LIN {X 0,Y 117.836,Z 740.059,A -85,B 0,C 180,E1 -26007.711,E2 -26007.711} C_VEL
LIN {X 0,Y 116.327,Z 745.047,A -85,B 0,C 180,E1 -26011.731,E2 -26011.731} C_VEL
LIN {X 0,Y 115.88,Z 750.752,A -85,B 0,C 180,E1 -26016.967,E2 -26016.967} C_VEL
LIN {X 0,Y 115.857,Z 756.729,A -85,B 0,C 180,E1 -26024.043,E2 -26024.043} C_VEL
LIN {X 0,Y 117.699,Z 761.437,A -85,B 0,C 180,E1 -26030.994,E2 -26030.994} C_VEL
LIN {X 0,Y 121.56,Z 765.132,A -85,B 0,C 180,E1 -26037.55,E2 -26037.55} C_VEL
LIN {X 0,Y 129.441,Z 768.589,A -85,B 0,C 180,E1 -26045.469,E2 -26045.469} C_VEL
LIN {X 0,Y 138.496,Z 770.335,A -85,B 0,C 180,E1 -26051.277,E2 -26051.277} C_VEL
LIN {X 0,Y 147.642,Z 770.918,A -85,B 0,C 180,E1 -26055.564,E2 -26055.564} C_VEL
LIN {X 0,Y 151.092,Z 770.908,A -85,B 0,C 180,E1 -26056.893,E2 -26056.893} C_VEL
LIN {X 0,Y 151.584,Z 770.825,A -85,B 0,C 180,E1 -26057.685,E2 -26057.685} C_VEL
LIN {X 0,Y 144.117,Z 770,A -85,B 0,C 180,E1 -26060.657,E2 -26060.657} C_VEL
LIN {X 0,Y 136.812,Z 768.361,A -85,B 0,C 180,E1 -26064.334,E2 -26064.334} C_VEL
LIN {X 0,Y 132.911,Z 767.253,A -85,B 0,C 180,E1 -26066.154,E2 -26066.154} C_VEL
LIN {X 0,Y 125.626,Z 764.718,A -85,B 0,C 180,E1 -26068.907,E2 -26068.907} C_VEL
LIN {X 0,Y 118.967,Z 761.486,A -85,B 0,C 180,E1 -26071.986,E2 -26071.986} C_VEL
LIN {X 0,Y 116.161,Z 759.416,A -85,B 0,C 180,E1 -26074.303,E2 -26074.303} C_VEL
LIN {X 0,Y 111.413,Z 753.187,A -85,B 0,C 180,E1 -26081.615,E2 -26081.615} C_VEL
LIN {X 0,Y 108.838,Z 744.994,A -85,B 0,C 180,E1 -26089.771,E2 -26089.771} C_VEL
LIN {X 0,Y 108.339,Z 738.209,A -85,B 0,C 180,E1 -26095.349,E2 -26095.349} C_VEL
LIN {X 0,Y 108.225,Z 729.961,A -85,B 0,C 180,E1 -26100.93,E2 -26100.93} C_VEL
LIN {X 0,Y 108.303,Z 721.553,A -85,B 0,C 180,E1 -26105.586,E2 -26105.586} C_VEL
LIN {X 0,Y 108.9,Z 710.32,A -85,B 0,C 180,E1 -26110.693,E2 -26110.693} C_VEL
LIN {X 0,Y 109.945,Z 696.049,A -85,B 0,C 180,E1 -26115.859,E2 -26115.859} C_VEL
LIN {X 0,Y 111.19,Z 683.821,A -85,B 0,C 180,E1 -26119.38,E2 -26119.38} C_VEL
LIN {X 0,Y 112.386,Z 671.062,A -85,B 0,C 180,E1 -26122.279,E2 -26122.279} C_VEL
LIN {X 0,Y 113.626,Z 656.475,A -85,B 0,C 180,E1 -26124.799,E2 -26124.799} C_VEL
LIN {X 0,Y 117.508,Z 604.417,A -85,B 0,C 180,E1 -26131.43,E2 -26131.43} C_VEL
LIN {X 0,Y 118.923,Z 587.439,A -85,B 0,C 180,E1 -26133.466,E2 -26133.466} C_VEL
LIN {X 0,Y 117.065,Z 560.293,A -85,B 0,C 180,E1 -26136.871,E2 -26136.871} C_VEL
LIN {X 0,Y 110.897,Z 536.307,A -85,B 0,C 180,E1 -26140.492,E2 -26140.492} C_VEL
LIN {X 0,Y 108.832,Z 527.055,A -85,B 0,C 180,E1 -26147.308,E2 -26147.308} C_VEL
LIN {X 0,Y 107.788,Z 522.184,A -85,B 0,C 180,E1 -26151.2,E2 -26151.2} C_VEL
LIN {X 0,Y 107.799,Z 522.181,A -85,B 0,C 180,E1 -26158.562,E2 -26158.562} C_VEL
LIN {X 0,Y 107.912,Z 522.166,A -85,B 0,C 180,E1 -26166.998,E2 -26166.998} C_VEL
LIN {X 0,Y 108.041,Z 522.149,A -85,B 0,C 180,E1 -26174.918,E2 -26174.918} C_VEL
LIN {X 0,Y 108.308,Z 522.117,A -85,B 0,C 180,E1 -26178.774,E2 -26178.774} C_VEL
LIN {X 0,Y 108.466,Z 522.098,A -85,B 0,C 180,E1 -26186.285,E2 -26186.285} C_VEL
LIN {X 0,Y 108.949,Z 522.032,A -85,B 0,C 180,E1 -26190,E2 -26190} C_VEL
LIN {X 0,Y 108.342,Z 522.108,A -85,B 0,C 180,E1 -26197.454,E2 -26197.454} C_VEL
LIN {X 0,Y 108.204,Z 522.132,A -85,B 0,C 180,E1 -26203.026,E2 -26203.026} C_VEL
LIN {X 0,Y 107.911,Z 522.165,A -85,B 0,C 180,E1 -26209.004,E2 -26209.004} C_VEL
LIN {X 0,Y 107.858,Z 522.169,A -85,B 0,C 180,E1 -26214.184,E2 -26214.184} C_VEL
LIN {X 0,Y 107.795,Z 522.179,A -85,B 0,C 180,E1 -26222.052,E2 -26222.052} C_VEL
LIN {X 0,Y 107.715,Z 522.192,A -85,B 0,C 180,E1 -26228.468,E2 -26228.468} C_VEL
LIN {X 0,Y 107.852,Z 522.23,A -85,B 0,C 180,E1 -26233.59,E2 -26233.59} C_VEL
LIN {X 0,Y 111.116,Z 536.487,A -85,B 0,C 180,E1 -26240.246,E2 -26240.246} C_VEL
LIN {X 0,Y 114.313,Z 550.66,A -85,B 0,C 180,E1 -26246.405,E2 -26246.405} C_VEL
LIN {X 0,Y 114.295,Z 554.161,A -85,B 0,C 180,E1 -26247.728,E2 -26247.728} C_VEL
LIN {X 0,Y 115.295,Z 578.296,A -85,B 0,C 180,E1 -26250.622,E2 -26250.622} C_VEL
LIN {X 0,Y 116.148,Z 589.056,A -85,B 0,C 180,E1 -26251.911,E2 -26251.911} C_VEL
LIN {X 0,Y 112.728,Z 655.949,A -85,B 0,C 180,E1 -26260.525,E2 -26260.525} C_VEL
LIN {X 0,Y 111.929,Z 671.773,A -85,B 0,C 180,E1 -26262.883,E2 -26262.883} C_VEL
LIN {X 0,Y 111.129,Z 684.001,A -85,B 0,C 180,E1 -26265.347,E2 -26265.347} C_VEL
LIN {X 0,Y 110.258,Z 697.634,A -85,B 0,C 180,E1 -26268.976,E2 -26268.976} C_VEL
LIN {X 0,Y 109.668,Z 708.586,A -85,B 0,C 180,E1 -26272.636,E2 -26272.636} C_VEL
LIN {X 0,Y 109.307,Z 719.724,A -85,B 0,C 180,E1 -26277.236,E2 -26277.236} C_VEL
LIN {X 0,Y 109.26,Z 728.724,A -85,B 0,C 180,E1 -26281.843,E2 -26281.843} C_VEL
LIN {X 0,Y 109.364,Z 736.128,A -85,B 0,C 180,E1 -26286.457,E2 -26286.457} C_VEL
LIN {X 0,Y 109.683,Z 743.345,A -85,B 0,C 180,E1 -26292.02,E2 -26292.02} C_VEL
LIN {X 0,Y 111.458,Z 750.421,A -85,B 0,C 180,E1 -26298.378,E2 -26298.378} C_VEL
LIN {X 0,Y 115.207,Z 756.964,A -85,B 0,C 180,E1 -26305.279,E2 -26305.279} C_VEL
LIN {X 0,Y 120.801,Z 762.203,A -85,B 0,C 180,E1 -26311.574,E2 -26311.574} C_VEL
LIN {X 0,Y 128.236,Z 766.306,A -85,B 0,C 180,E1 -26317.075,E2 -26317.075} C_VEL
LIN {X 0,Y 137.135,Z 769.302,A -85,B 0,C 180,E1 -26321.777,E2 -26321.777} C_VEL
LIN {X 0,Y 140.576,Z 770.083,A -85,B 0,C 180,E1 -26323.232,E2 -26323.232} C_VEL
LIN {X 0,Y 140.221,Z 770.131,A -85,B 0,C 180,E1 -26324.287,E2 -26324.287} C_VEL
LIN {X 0,Y 129.693,Z 768.061,A -85,B 0,C 180,E1 -26329.438,E2 -26329.438} C_VEL
LIN {X 0,Y 122.094,Z 765.265,A -85,B 0,C 180,E1 -26334.857,E2 -26334.857} C_VEL
LIN {X 0,Y 116.195,Z 761.467,A -85,B 0,C 180,E1 -26341.061,E2 -26341.061} C_VEL
LIN {X 0,Y 112.25,Z 756.576,A -85,B 0,C 180,E1 -26347.935,E2 -26347.935} C_VEL
LIN {X 0,Y 110.479,Z 750.464,A -85,B 0,C 180,E1 -26355.259,E2 -26355.259} C_VEL
LIN {X 0,Y 110.594,Z 743.772,A -85,B 0,C 180,E1 -26361.78,E2 -26361.78} C_VEL
LIN {X 0,Y 111.699,Z 736.584,A -85,B 0,C 180,E1 -26367.45,E2 -26367.45} C_VEL
LIN {X 0,Y 109.948,Z 741.833,A -85,B 0,C 180,E1 -26371.832,E2 -26371.832} C_VEL
LIN {X 0,Y 109.438,Z 747.875,A -85,B 0,C 180,E1 -26377.38,E2 -26377.38} C_VEL
LIN {X 0,Y 109.482,Z 754.136,A -85,B 0,C 180,E1 -26384.879,E2 -26384.879} C_VEL
LIN {X 0,Y 111.446,Z 759.184,A -85,B 0,C 180,E1 -26392.233,E2 -26392.233} C_VEL
LIN {X 0,Y 115.538,Z 763.209,A -85,B 0,C 180,E1 -26399.119,E2 -26399.119} C_VEL
LIN {X 0,Y 121.444,Z 766.263,A -85,B 0,C 180,E1 -26405.36,E2 -26405.36} C_VEL
LIN {X 0,Y 129.062,Z 768.493,A -85,B 0,C 180,E1 -26410.803,E2 -26410.803} C_VEL
LIN {X 0,Y 139.931,Z 770.054,A -85,B 0,C 180,E1 -26416.427,E2 -26416.427} C_VEL
LIN {X 0,Y 141.036,Z 770.146,A -85,B 0,C 180,E1 -26416.878,E2 -26416.878} C_VEL
LIN {X 0,Y 140.5,Z 769.925,A -85,B 0,C 180,E1 -26418.058,E2 -26418.058} C_VEL
LIN {X 0,Y 129.613,Z 767.124,A -85,B 0,C 180,E1 -26423.384,E2 -26423.384} C_VEL
LIN {X 0,Y 120.074,Z 762.583,A -85,B 0,C 180,E1 -26430.164,E2 -26430.164} C_VEL
LIN {X 0,Y 116.161,Z 759.416,A -85,B 0,C 180,E1 -26434.303,E2 -26434.303} C_VEL
LIN {X 0,Y 113.641,Z 757.196,A -85,B 0,C 180,E1 -26436.712,E2 -26436.712} C_VEL
LIN {X 0,Y 106.531,Z 750.669,A -85,B 0,C 180,E1 -26441.919,E2 -26441.919} C_VEL
LIN {X 0,Y 103.471,Z 746.464,A -85,B 0,C 180,E1 -26445.213,E2 -26445.213} C_VEL
LIN {X 0,Y 102.733,Z 744.402,A -85,B 0,C 180,E1 -26447.052,E2 -26447.052} C_VEL
LIN {X 0,Y 101.854,Z 736.413,A -85,B 0,C 180,E1 -26454.059,E2 -26454.059} C_VEL
LIN {X 0,Y 101.623,Z 729.435,A -85,B 0,C 180,E1 -26459.009,E2 -26459.009} C_VEL
LIN {X 0,Y 101.655,Z 721.117,A -85,B 0,C 180,E1 -26463.964,E2 -26463.964} C_VEL
LIN {X 0,Y 102.025,Z 710.024,A -85,B 0,C 180,E1 -26469.416,E2 -26469.416} C_VEL
LIN {X 0,Y 102.767,Z 697.76,A -85,B 0,C 180,E1 -26474.209,E2 -26474.209} C_VEL
LIN {X 0,Y 103.928,Z 686.164,A -85,B 0,C 180,E1 -26477.938,E2 -26477.938} C_VEL
LIN {X 0,Y 105.202,Z 672.771,A -85,B 0,C 180,E1 -26481.351,E2 -26481.351} C_VEL
LIN {X 0,Y 106.464,Z 657.142,A -85,B 0,C 180,E1 -26484.367,E2 -26484.367} C_VEL
LIN {X 0,Y 109.13,Z 620.339,A -85,B 0,C 180,E1 -26489.542,E2 -26489.542} C_VEL
LIN {X 0,Y 111.81,Z 587.596,A -85,B 0,C 180,E1 -26493.772,E2 -26493.772} C_VEL
LIN {X 0,Y 110.129,Z 561.697,A -85,B 0,C 180,E1 -26497.239,E2 -26497.239} C_VEL
LIN {X 0,Y 103.597,Z 536.147,A -85,B 0,C 180,E1 -26501.368,E2 -26501.368} C_VEL
LIN {X 0,Y 101.86,Z 528.349,A -85,B 0,C 180,E1 -26507.502,E2 -26507.502} C_VEL
LIN {X 0,Y 100.703,Z 523.066,A -85,B 0,C 180,E1 -26512.046,E2 -26512.046} C_VEL
LIN {X 0,Y 100.693,Z 523.062,A -85,B 0,C 180,E1 -26516.882,E2 -26516.882} C_VEL
LIN {X 0,Y 100.787,Z 523.049,A -85,B 0,C 180,E1 -26525.267,E2 -26525.267} C_VEL
LIN {X 0,Y 100.82,Z 523.051,A -85,B 0,C 180,E1 -26529.601,E2 -26529.601} C_VEL
LIN {X 0,Y 101.2,Z 523.003,A -85,B 0,C 180,E1 -26537.975,E2 -26537.975} C_VEL
LIN {X 0,Y 101.281,Z 522.988,A -85,B 0,C 180,E1 -26542.022,E2 -26542.022} C_VEL
LIN {X 0,Y 101.873,Z 522.913,A -85,B 0,C 180,E1 -26550,E2 -26550} C_VEL
LIN {X 0,Y 101.281,Z 522.986,A -85,B 0,C 180,E1 -26557.977,E2 -26557.977} C_VEL
LIN {X 0,Y 101.13,Z 523.013,A -85,B 0,C 180,E1 -26563.363,E2 -26563.363} C_VEL
LIN {X 0,Y 100.82,Z 523.051,A -85,B 0,C 180,E1 -26570.398,E2 -26570.398} C_VEL
LIN {X 0,Y 100.775,Z 523.05,A -85,B 0,C 180,E1 -26574.958,E2 -26574.958} C_VEL
LIN {X 0,Y 100.701,Z 523.06,A -85,B 0,C 180,E1 -26583.124,E2 -26583.124} C_VEL
LIN {X 0,Y 100.739,Z 523.053,A -85,B 0,C 180,E1 -26591.798,E2 -26591.798} C_VEL
LIN {X 0,Y 100.813,Z 523.12,A -85,B 0,C 180,E1 -26592.967,E2 -26592.967} C_VEL
LIN {X 0,Y 104.128,Z 537.755,A -85,B 0,C 180,E1 -26600.152,E2 -26600.152} C_VEL
LIN {X 0,Y 107.067,Z 550.686,A -85,B 0,C 180,E1 -26606.088,E2 -26606.088} C_VEL
LIN {X 0,Y 107.21,Z 553.958,A -85,B 0,C 180,E1 -26607.472,E2 -26607.472} C_VEL
LIN {X 0,Y 108.263,Z 579.215,A -85,B 0,C 180,E1 -26610.75,E2 -26610.75} C_VEL
LIN {X 0,Y 108.966,Z 589.885,A -85,B 0,C 180,E1 -26612.121,E2 -26612.121} C_VEL
LIN {X 0,Y 105.725,Z 658.101,A -85,B 0,C 180,E1 -26621.594,E2 -26621.594} C_VEL
LIN {X 0,Y 104.911,Z 673.601,A -85,B 0,C 180,E1 -26624.208,E2 -26624.208} C_VEL
LIN {X 0,Y 104.067,Z 687.071,A -85,B 0,C 180,E1 -26627.321,E2 -26627.321} C_VEL
LIN {X 0,Y 103.38,Z 700.092,A -85,B 0,C 180,E1 -26631.202,E2 -26631.202} C_VEL
LIN {X 0,Y 102.914,Z 710.414,A -85,B 0,C 180,E1 -26635.103,E2 -26635.103} C_VEL
LIN {X 0,Y 102.837,Z 721.004,A -85,B 0,C 180,E1 -26640,E2 -26640} C_VEL
LIN {X 0,Y 102.956,Z 729.651,A -85,B 0,C 180,E1 -26644.895,E2 -26644.895} C_VEL
LIN {X 0,Y 103.139,Z 736.605,A -85,B 0,C 180,E1 -26649.808,E2 -26649.808} C_VEL
LIN {X 0,Y 104.524,Z 745.743,A -85,B 0,C 180,E1 -26657.612,E2 -26657.612} C_VEL
LIN {X 0,Y 107.965,Z 753.091,A -85,B 0,C 180,E1 -26665.032,E2 -26665.032} C_VEL
LIN {X 0,Y 113.43,Z 759.062,A -85,B 0,C 180,E1 -26671.779,E2 -26671.779} C_VEL
LIN {X 0,Y 120.684,Z 763.854,A -85,B 0,C 180,E1 -26677.696,E2 -26677.696} C_VEL
LIN {X 0,Y 130.665,Z 767.952,A -85,B 0,C 180,E1 -26683.202,E2 -26683.202} C_VEL
LIN {X 0,Y 130.428,Z 768.003,A -85,B 0,C 180,E1 -26684.327,E2 -26684.327} C_VEL
LIN {X 0,Y 124.527,Z 766.414,A -85,B 0,C 180,E1 -26687.371,E2 -26687.371} C_VEL
LIN {X 0,Y 116.607,Z 763.235,A -85,B 0,C 180,E1 -26692.936,E2 -26692.936} C_VEL
LIN {X 0,Y 110.417,Z 759.069,A -85,B 0,C 180,E1 -26699.39,E2 -26699.39} C_VEL
LIN {X 0,Y 106.233,Z 753.781,A -85,B 0,C 180,E1 -26706.613,E2 -26706.613} C_VEL
LIN {X 0,Y 104.358,Z 747.267,A -85,B 0,C 180,E1 -26714.373,E2 -26714.373} C_VEL
LIN {X 0,Y 104.382,Z 741.354,A -85,B 0,C 180,E1 -26720.31,E2 -26720.31} C_VEL
LIN {X 0,Y 105.663,Z 732.897,A -85,B 0,C 180,E1 -26727.248,E2 -26727.248} C_VEL
LIN {X 0,Y 103.663,Z 738.443,A -85,B 0,C 180,E1 -26731.943,E2 -26731.943} C_VEL
LIN {X 0,Y 103.087,Z 744.796,A -85,B 0,C 180,E1 -26737.837,E2 -26737.837} C_VEL
LIN {X 0,Y 103.171,Z 751.383,A -85,B 0,C 180,E1 -26745.812,E2 -26745.812} C_VEL
LIN {X 0,Y 105.317,Z 756.697,A -85,B 0,C 180,E1 -26753.603,E2 -26753.603} C_VEL
LIN {X 0,Y 109.681,Z 761.067,A -85,B 0,C 180,E1 -26760.839,E2 -26760.839} C_VEL
LIN {X 0,Y 115.909,Z 764.481,A -85,B 0,C 180,E1 -26767.326,E2 -26767.326} C_VEL
LIN {X 0,Y 123.89,Z 767.035,A -85,B 0,C 180,E1 -26772.902,E2 -26772.902} C_VEL
LIN {X 0,Y 131.226,Z 768.538,A -85,B 0,C 180,E1 -26776.85,E2 -26776.85} C_VEL
LIN {X 0,Y 130.525,Z 768.205,A -85,B 0,C 180,E1 -26778.142,E2 -26778.142} C_VEL
LIN {X 0,Y 119.793,Z 764.229,A -85,B 0,C 180,E1 -26784.078,E2 -26784.078} C_VEL
LIN {X 0,Y 112.489,Z 759.76,A -85,B 0,C 180,E1 -26790.012,E2 -26790.012} C_VEL
LIN {X 0,Y 107.088,Z 754.177,A -85,B 0,C 180,E1 -26796.811,E2 -26796.811} C_VEL
LIN {X 0,Y 103.505,Z 747.281,A -85,B 0,C 180,E1 -26804.24,E2 -26804.24} C_VEL
LIN {X 0,Y 102.733,Z 744.402,A -85,B 0,C 180,E1 -26807.052,E2 -26807.052} C_VEL
LIN {X 0,Y 101.66,Z 741.184,A -85,B 0,C 180,E1 -26809.735,E2 -26809.735} C_VEL
LIN {X 0,Y 99.905,Z 737.51,A -85,B 0,C 180,E1 -26812.19,E2 -26812.19} C_VEL
LIN {X 0,Y 96.165,Z 729.337,A -85,B 0,C 180,E1 -26816.906,E2 -26816.906} C_VEL
LIN {X 0,Y 95.15,Z 725.073,A -85,B 0,C 180,E1 -26819.392,E2 -26819.392} C_VEL
LIN {X 0,Y 95.071,Z 723.636,A -85,B 0,C 180,E1 -26820.254,E2 -26820.254} C_VEL
LIN {X 0,Y 95.168,Z 713.731,A -85,B 0,C 180,E1 -26825.828,E2 -26825.828} C_VEL
LIN {X 0,Y 95.538,Z 703.495,A -85,B 0,C 180,E1 -26830.597,E2 -26830.597} C_VEL
LIN {X 0,Y 96.562,Z 689.721,A -85,B 0,C 180,E1 -26835.839,E2 -26835.839} C_VEL
LIN {X 0,Y 97.905,Z 675.435,A -85,B 0,C 180,E1 -26840.001,E2 -26840.001} C_VEL
LIN {X 0,Y 99.236,Z 659.449,A -85,B 0,C 180,E1 -26843.474,E2 -26843.474} C_VEL
LIN {X 0,Y 101.423,Z 628.397,A -85,B 0,C 180,E1 -26848.309,E2 -26848.309} C_VEL
LIN {X 0,Y 104.746,Z 588.113,A -85,B 0,C 180,E1 -26854.047,E2 -26854.047} C_VEL
LIN {X 0,Y 103.146,Z 562.959,A -85,B 0,C 180,E1 -26857.63,E2 -26857.63} C_VEL
LIN {X 0,Y 96.32,Z 536.044,A -85,B 0,C 180,E1 -26862.261,E2 -26862.261} C_VEL
LIN {X 0,Y 94.467,Z 527.663,A -85,B 0,C 180,E1 -26869.385,E2 -26869.385} C_VEL
LIN {X 0,Y 93.655,Z 523.943,A -85,B 0,C 180,E1 -26872.769,E2 -26872.769} C_VEL
LIN {X 0,Y 93.585,Z 523.952,A -85,B 0,C 180,E1 -26878.285,E2 -26878.285} C_VEL
LIN {X 0,Y 93.67,Z 523.934,A -85,B 0,C 180,E1 -26884.205,E2 -26884.205} C_VEL
LIN {X 0,Y 93.696,Z 523.939,A -85,B 0,C 180,E1 -26887.973,E2 -26887.973} C_VEL
LIN {X 0,Y 94.099,Z 523.889,A -85,B 0,C 180,E1 -26897.052,E2 -26897.052} C_VEL
LIN {X 0,Y 94.213,Z 523.867,A -85,B 0,C 180,E1 -26901.419,E2 -26901.419} C_VEL
LIN {X 0,Y 94.8,Z 523.794,A -85,B 0,C 180,E1 -26910,E2 -26910} C_VEL
LIN {X 0,Y 94.213,Z 523.866,A -85,B 0,C 180,E1 -26918.58,E2 -26918.58} C_VEL
LIN {X 0,Y 94.048,Z 523.894,A -85,B 0,C 180,E1 -26923.721,E2 -26923.721} C_VEL
LIN {X 0,Y 93.696,Z 523.938,A -85,B 0,C 180,E1 -26932.027,E2 -26932.027} C_VEL
LIN {X 0,Y 93.624,Z 523.943,A -85,B 0,C 180,E1 -26936.769,E2 -26936.769} C_VEL
LIN {X 0,Y 93.6,Z 523.944,A -85,B 0,C 180,E1 -26944.316,E2 -26944.316} C_VEL
LIN {X 0,Y 93.719,Z 523.931,A -85,B 0,C 180,E1 -26952.264,E2 -26952.264} C_VEL
LIN {X 0,Y 96.683,Z 537.098,A -85,B 0,C 180,E1 -26959.139,E2 -26959.139} C_VEL
LIN {X 0,Y 99.512,Z 549.365,A -85,B 0,C 180,E1 -26965.153,E2 -26965.153} C_VEL
LIN {X 0,Y 100.183,Z 553.098,A -85,B 0,C 180,E1 -26966.887,E2 -26966.887} C_VEL
LIN {X 0,Y 100.132,Z 554.433,A -85,B 0,C 180,E1 -26967.378,E2 -26967.378} C_VEL
LIN {X 0,Y 101.192,Z 579.73,A -85,B 0,C 180,E1 -26970.863,E2 -26970.863} C_VEL
LIN {X 0,Y 101.869,Z 589.828,A -85,B 0,C 180,E1 -26972.247,E2 -26972.247} C_VEL
LIN {X 0,Y 98.822,Z 657.872,A -85,B 0,C 180,E1 -26982.541,E2 -26982.541} C_VEL
LIN {X 0,Y 98.096,Z 672.774,A -85,B 0,C 180,E1 -26985.213,E2 -26985.213} C_VEL
LIN {X 0,Y 97.309,Z 686.365,A -85,B 0,C 180,E1 -26988.544,E2 -26988.544} C_VEL
LIN {X 0,Y 96.763,Z 699.268,A -85,B 0,C 180,E1 -26992.698,E2 -26992.698} C_VEL
LIN {X 0,Y 96.452,Z 710.8,A -85,B 0,C 180,E1 -26997.39,E2 -26997.39} C_VEL
LIN {X 0,Y 96.505,Z 720.267,A -85,B 0,C 180,E1 -27002.087,E2 -27002.087} C_VEL
LIN {X 0,Y 96.78,Z 728.722,A -85,B 0,C 180,E1 -27007.301,E2 -27007.301} C_VEL
LIN {X 0,Y 97.095,Z 735.657,A -85,B 0,C 180,E1 -27012.542,E2 -27012.542} C_VEL
LIN {X 0,Y 99.145,Z 744.746,A -85,B 0,C 180,E1 -27020.759,E2 -27020.759} C_VEL
LIN {X 0,Y 103.279,Z 752.18,A -85,B 0,C 180,E1 -27028.447,E2 -27028.447} C_VEL
LIN {X 0,Y 109.441,Z 758.277,A -85,B 0,C 180,E1 -27035.307,E2 -27035.307} C_VEL
LIN {X 0,Y 117.488,Z 763.257,A -85,B 0,C 180,E1 -27041.148,E2 -27041.148} C_VEL
LIN {X 0,Y 122.102,Z 765.337,A -85,B 0,C 180,E1 -27043.686,E2 -27043.686} C_VEL
LIN {X 0,Y 111.338,Z 760.936,A -85,B 0,C 180,E1 -27050.859,E2 -27050.859} C_VEL
LIN {X 0,Y 104.828,Z 756.384,A -85,B 0,C 180,E1 -27057.565,E2 -27057.565} C_VEL
LIN {X 0,Y 100.394,Z 750.743,A -85,B 0,C 180,E1 -27065.164,E2 -27065.164} C_VEL
LIN {X 0,Y 98.367,Z 743.863,A -85,B 0,C 180,E1 -27073.394,E2 -27073.394} C_VEL
LIN {X 0,Y 98.345,Z 737.656,A -85,B 0,C 180,E1 -27079.709,E2 -27079.709} C_VEL
LIN {X 0,Y 99.77,Z 728.982,A -85,B 0,C 180,E1 -27086.973,E2 -27086.973} C_VEL
LIN {X 0,Y 97.742,Z 733.689,A -85,B 0,C 180,E1 -27091.03,E2 -27091.03} C_VEL
LIN {X 0,Y 96.839,Z 741.459,A -85,B 0,C 180,E1 -27098.346,E2 -27098.346} C_VEL
LIN {X 0,Y 96.975,Z 748.434,A -85,B 0,C 180,E1 -27106.852,E2 -27106.852} C_VEL
LIN {X 0,Y 100.275,Z 755.33,A -85,B 0,C 180,E1 -27117.102,E2 -27117.102} C_VEL
LIN {X 0,Y 107.043,Z 760.672,A -85,B 0,C 180,E1 -27126.221,E2 -27126.221} C_VEL
LIN {X 0,Y 115.631,Z 764.362,A -85,B 0,C 180,E1 -27133.167,E2 -27133.167} C_VEL
LIN {X 0,Y 120.76,Z 765.879,A -85,B 0,C 180,E1 -27136.232,E2 -27136.232} C_VEL
LIN {X 0,Y 121.87,Z 766.021,A -85,B 0,C 180,E1 -27137.674,E2 -27137.674} C_VEL
LIN {X 0,Y 112.177,Z 761.63,A -85,B 0,C 180,E1 -27143.474,E2 -27143.474} C_VEL
LIN {X 0,Y 103.543,Z 755.043,A -85,B 0,C 180,E1 -27151.632,E2 -27151.632} C_VEL
LIN {X 0,Y 98.794,Z 748.402,A -85,B 0,C 180,E1 -27159.164,E2 -27159.164} C_VEL
LIN {X 0,Y 96.146,Z 740.353,A -85,B 0,C 180,E1 -27167.332,E2 -27167.332} C_VEL
LIN {X 0,Y 95.439,Z 733.067,A -85,B 0,C 180,E1 -27173.658,E2 -27173.658} C_VEL
LIN {X 0,Y 95.152,Z 725.767,A -85,B 0,C 180,E1 -27178.942,E2 -27178.942} C_VEL
LIN {X 0,Y 95.071,Z 723.636,A -85,B 0,C 180,E1 -27180.254,E2 -27180.254} C_VEL
LIN {X 0,Y 94.476,Z 719.339,A -85,B 0,C 180,E1 -27182.608,E2 -27182.608} C_VEL
LIN {X 0,Y 93.062,Z 714.702,A -85,B 0,C 180,E1 -27184.679,E2 -27184.679} C_VEL
LIN {X 0,Y 89.786,Z 704.816,A -85,B 0,C 180,E1 -27188.498,E2 -27188.498} C_VEL
LIN {X 0,Y 88.986,Z 699.709,A -85,B 0,C 180,E1 -27190.508,E2 -27190.508} C_VEL
LIN {X 0,Y 88.988,Z 697.984,A -85,B 0,C 180,E1 -27191.214,E2 -27191.214} C_VEL
LIN {X 0,Y 89.977,Z 685.808,A -85,B 0,C 180,E1 -27195.865,E2 -27195.865} C_VEL
LIN {X 0,Y 91.176,Z 672.363,A -85,B 0,C 180,E1 -27199.904,E2 -27199.904} C_VEL
LIN {X 0,Y 92.333,Z 657.161,A -85,B 0,C 180,E1 -27203.345,E2 -27203.345} C_VEL
LIN {X 0,Y 94.975,Z 619.674,A -85,B 0,C 180,E1 -27209.508,E2 -27209.508} C_VEL
LIN {X 0,Y 97.641,Z 587.995,A -85,B 0,C 180,E1 -27214.314,E2 -27214.314} C_VEL
LIN {X 0,Y 96.148,Z 564.258,A -85,B 0,C 180,E1 -27217.955,E2 -27217.955} C_VEL
LIN {X 0,Y 89.035,Z 535.943,A -85,B 0,C 180,E1 -27223.204,E2 -27223.204} C_VEL
LIN {X 0,Y 87.139,Z 527.353,A -85,B 0,C 180,E1 -27231.137,E2 -27231.137} C_VEL
LIN {X 0,Y 86.578,Z 524.821,A -85,B 0,C 180,E1 -27233.858,E2 -27233.858} C_VEL
LIN {X 0,Y 86.585,Z 524.818,A -85,B 0,C 180,E1 -27243.234,E2 -27243.234} C_VEL
LIN {X 0,Y 86.665,Z 524.81,A -85,B 0,C 180,E1 -27251.072,E2 -27251.072} C_VEL
LIN {X 0,Y 86.97,Z 524.777,A -85,B 0,C 180,E1 -27255.97,E2 -27255.97} C_VEL
LIN {X 0,Y 87.119,Z 524.75,A -85,B 0,C 180,E1 -27260.715,E2 -27260.715} C_VEL
LIN {X 0,Y 87.727,Z 524.675,A -85,B 0,C 180,E1 -27270,E2 -27270} C_VEL
LIN {X 0,Y 87.119,Z 524.751,A -85,B 0,C 180,E1 -27279.285,E2 -27279.285} C_VEL
LIN {X 0,Y 86.951,Z 524.777,A -85,B 0,C 180,E1 -27284.087,E2 -27284.087} C_VEL
LIN {X 0,Y 86.667,Z 524.811,A -85,B 0,C 180,E1 -27288.927,E2 -27288.927} C_VEL
LIN {X 0,Y 86.586,Z 524.82,A -85,B 0,C 180,E1 -27296.767,E2 -27296.767} C_VEL
LIN {X 0,Y 86.521,Z 524.829,A -85,B 0,C 180,E1 -27305.68,E2 -27305.68} C_VEL
LIN {X 0,Y 86.624,Z 524.812,A -85,B 0,C 180,E1 -27311.528,E2 -27311.528} C_VEL
LIN {X 0,Y 89.646,Z 538.148,A -85,B 0,C 180,E1 -27318.988,E2 -27318.988} C_VEL
LIN {X 0,Y 92.34,Z 549.631,A -85,B 0,C 180,E1 -27324.945,E2 -27324.945} C_VEL
LIN {X 0,Y 93.045,Z 554.146,A -85,B 0,C 180,E1 -27327.17,E2 -27327.17} C_VEL
LIN {X 0,Y 94.128,Z 580.203,A -85,B 0,C 180,E1 -27331.106,E2 -27331.106} C_VEL
LIN {X 0,Y 94.792,Z 589.437,A -85,B 0,C 180,E1 -27332.474,E2 -27332.474} C_VEL
LIN {X 0,Y 92.043,Z 653.392,A -85,B 0,C 180,E1 -27342.933,E2 -27342.933} C_VEL
LIN {X 0,Y 91.408,Z 670.341,A -85,B 0,C 180,E1 -27346.098,E2 -27346.098} C_VEL
LIN {X 0,Y 90.791,Z 683.378,A -85,B 0,C 180,E1 -27349.406,E2 -27349.406} C_VEL
LIN {X 0,Y 90.348,Z 695.395,A -85,B 0,C 180,E1 -27353.299,E2 -27353.299} C_VEL
LIN {X 0,Y 90.077,Z 706.314,A -85,B 0,C 180,E1 -27357.764,E2 -27357.764} C_VEL
LIN {X 0,Y 90.274,Z 715.349,A -85,B 0,C 180,E1 -27362.231,E2 -27362.231} C_VEL
LIN {X 0,Y 90.644,Z 724.553,A -85,B 0,C 180,E1 -27367.798,E2 -27367.798} C_VEL
LIN {X 0,Y 90.99,Z 730.576,A -85,B 0,C 180,E1 -27372.264,E2 -27372.264} C_VEL
LIN {X 0,Y 92.81,Z 740.449,A -85,B 0,C 180,E1 -27381.081,E2 -27381.081} C_VEL
LIN {X 0,Y 97.583,Z 749.42,A -85,B 0,C 180,E1 -27390.275,E2 -27390.275} C_VEL
LIN {X 0,Y 104.054,Z 755.914,A -85,B 0,C 180,E1 -27397.436,E2 -27397.436} C_VEL
LIN {X 0,Y 112.443,Z 761.315,A -85,B 0,C 180,E1 -27403.435,E2 -27403.435} C_VEL
LIN {X 0,Y 110.409,Z 760.5,A -85,B 0,C 180,E1 -27405.557,E2 -27405.557} C_VEL
LIN {X 0,Y 100.964,Z 754.83,A -85,B 0,C 180,E1 -27413.724,E2 -27413.724} C_VEL
LIN {X 0,Y 94.701,Z 747.495,A -85,B 0,C 180,E1 -27423.559,E2 -27423.559} C_VEL
LIN {X 0,Y 92.434,Z 739.24,A -85,B 0,C 180,E1 -27433.434,E2 -27433.434} C_VEL
LIN {X 0,Y 92.516,Z 733.411,A -85,B 0,C 180,E1 -27439.274,E2 -27439.274} C_VEL
LIN {X 0,Y 93.652,Z 725.765,A -85,B 0,C 180,E1 -27445.697,E2 -27445.697} C_VEL
LIN {X 0,Y 94.068,Z 724.766,A -85,B 0,C 180,E1 -27446.57,E2 -27446.57} C_VEL
LIN {X 0,Y 91.721,Z 729.775,A -85,B 0,C 180,E1 -27451.113,E2 -27451.113} C_VEL
LIN {X 0,Y 90.654,Z 738.944,A -85,B 0,C 180,E1 -27460.046,E2 -27460.046} C_VEL
LIN {X 0,Y 90.94,Z 745.213,A -85,B 0,C 180,E1 -27468.007,E2 -27468.007} C_VEL
LIN {X 0,Y 93.48,Z 751.18,A -85,B 0,C 180,E1 -27476.814,E2 -27476.814} C_VEL
LIN {X 0,Y 100.04,Z 757.258,A -85,B 0,C 180,E1 -27486.666,E2 -27486.666} C_VEL
LIN {X 0,Y 109.639,Z 761.927,A -85,B 0,C 180,E1 -27494.84,E2 -27494.84} C_VEL
LIN {X 0,Y 112.417,Z 762.888,A -85,B 0,C 180,E1 -27496.552,E2 -27496.552} C_VEL
LIN {X 0,Y 108.906,Z 760.989,A -85,B 0,C 180,E1 -27499.81,E2 -27499.81} C_VEL
LIN {X 0,Y 100.943,Z 755.742,A -85,B 0,C 180,E1 -27506.152,E2 -27506.152} C_VEL
LIN {X 0,Y 94.937,Z 749.398,A -85,B 0,C 180,E1 -27513.63,E2 -27513.63} C_VEL
LIN {X 0,Y 90.99,Z 741.629,A -85,B 0,C 180,E1 -27522.003,E2 -27522.003} C_VEL
LIN {X 0,Y 89.383,Z 733.549,A -85,B 0,C 180,E1 -27529.81,E2 -27529.81} C_VEL
LIN {X 0,Y 88.887,Z 726.5,A -85,B 0,C 180,E1 -27535.465,E2 -27535.465} C_VEL
LIN {X 0,Y 88.577,Z 718.02,A -85,B 0,C 180,E1 -27541.136,E2 -27541.136} C_VEL
LIN {X 0,Y 88.678,Z 707.673,A -85,B 0,C 180,E1 -27546.827,E2 -27546.827} C_VEL
LIN {X 0,Y 88.988,Z 697.984,A -85,B 0,C 180,E1 -27551.214,E2 -27551.214} C_VEL
LIN {X 0,Y 88.686,Z 692.895,A -85,B 0,C 180,E1 -27553.13,E2 -27553.13} C_VEL
LIN {X 0,Y 86.696,Z 684.059,A -85,B 0,C 180,E1 -27555.764,E2 -27555.764} C_VEL
LIN {X 0,Y 84.97,Z 676.782,A -85,B 0,C 180,E1 -27557.675,E2 -27557.675} C_VEL
LIN {X 0,Y 84.346,Z 671.237,A -85,B 0,C 180,E1 -27559.121,E2 -27559.121} C_VEL
LIN {X 0,Y 84.366,Z 669.383,A -85,B 0,C 180,E1 -27559.614,E2 -27559.614} C_VEL
LIN {X 0,Y 85.542,Z 653.688,A -85,B 0,C 180,E1 -27563.235,E2 -27563.235} C_VEL
LIN {X 0,Y 89.049,Z 605.004,A -85,B 0,C 180,E1 -27571.857,E2 -27571.857} C_VEL
LIN {X 0,Y 90.54,Z 588.123,A -85,B 0,C 180,E1 -27574.584,E2 -27574.584} C_VEL
LIN {X 0,Y 89.071,Z 565.15,A -85,B 0,C 180,E1 -27578.407,E2 -27578.407} C_VEL
LIN {X 0,Y 81.74,Z 535.783,A -85,B 0,C 180,E1 -27584.312,E2 -27584.312} C_VEL
LIN {X 0,Y 79.998,Z 527.88,A -85,B 0,C 180,E1 -27592.248,E2 -27592.248} C_VEL
LIN {X 0,Y 79.521,Z 525.698,A -85,B 0,C 180,E1 -27594.778,E2 -27594.778} C_VEL
LIN {X 0,Y 79.526,Z 525.696,A -85,B 0,C 180,E1 -27603.776,E2 -27603.776} C_VEL
LIN {X 0,Y 79.524,Z 525.704,A -85,B 0,C 180,E1 -27609.298,E2 -27609.298} C_VEL
LIN {X 0,Y 79.842,Z 525.663,A -85,B 0,C 180,E1 -27615.525,E2 -27615.525} C_VEL
LIN {X 0,Y 80.002,Z 525.639,A -85,B 0,C 180,E1 -27619.88,E2 -27619.88} C_VEL
LIN {X 0,Y 80.655,Z 525.555,A -85,B 0,C 180,E1 -27630,E2 -27630} C_VEL
LIN {X 0,Y 80.001,Z 525.641,A -85,B 0,C 180,E1 -27640.119,E2 -27640.119} C_VEL
LIN {X 0,Y 79.767,Z 525.668,A -85,B 0,C 180,E1 -27645.326,E2 -27645.326} C_VEL
LIN {X 0,Y 79.525,Z 525.704,A -85,B 0,C 180,E1 -27650.701,E2 -27650.701} C_VEL
LIN {X 0,Y 79.484,Z 525.708,A -85,B 0,C 180,E1 -27657.846,E2 -27657.846} C_VEL
LIN {X 0,Y 79.44,Z 525.714,A -85,B 0,C 180,E1 -27667.23,E2 -27667.23} C_VEL
LIN {X 0,Y 79.556,Z 525.823,A -85,B 0,C 180,E1 -27670.864,E2 -27670.864} C_VEL
LIN {X 0,Y 82.15,Z 536.904,A -85,B 0,C 180,E1 -27677.55,E2 -27677.55} C_VEL
LIN {X 0,Y 85.099,Z 549.688,A -85,B 0,C 180,E1 -27684.683,E2 -27684.683} C_VEL
LIN {X 0,Y 85.976,Z 554.105,A -85,B 0,C 180,E1 -27687.037,E2 -27687.037} C_VEL
LIN {X 0,Y 86.905,Z 578.497,A -85,B 0,C 180,E1 -27691.067,E2 -27691.067} C_VEL
LIN {X 0,Y 87.682,Z 589.954,A -85,B 0,C 180,E1 -27692.893,E2 -27692.893} C_VEL
LIN {X 0,Y 85.26,Z 652.464,A -85,B 0,C 180,E1 -27704.154,E2 -27704.154} C_VEL
LIN {X 0,Y 84.734,Z 670.183,A -85,B 0,C 180,E1 -27707.729,E2 -27707.729} C_VEL
LIN {X 0,Y 84.231,Z 682.231,A -85,B 0,C 180,E1 -27711,E2 -27711} C_VEL
LIN {X 0,Y 83.953,Z 694.206,A -85,B 0,C 180,E1 -27715.198,E2 -27715.198} C_VEL
LIN {X 0,Y 83.9,Z 705.18,A -85,B 0,C 180,E1 -27720,E2 -27720} C_VEL
LIN {X 0,Y 84.235,Z 714.273,A -85,B 0,C 180,E1 -27724.786,E2 -27724.786} C_VEL
LIN {X 0,Y 84.727,Z 721.716,A -85,B 0,C 180,E1 -27729.55,E2 -27729.55} C_VEL
LIN {X 0,Y 85.202,Z 727.882,A -85,B 0,C 180,E1 -27734.327,E2 -27734.327} C_VEL
LIN {X 0,Y 87.049,Z 736.854,A -85,B 0,C 180,E1 -27742.551,E2 -27742.551} C_VEL
LIN {X 0,Y 90.745,Z 744.493,A -85,B 0,C 180,E1 -27750.353,E2 -27750.353} C_VEL
LIN {X 0,Y 97.051,Z 751.665,A -85,B 0,C 180,E1 -27757.991,E2 -27757.991} C_VEL
LIN {X 0,Y 104.157,Z 757.007,A -85,B 0,C 180,E1 -27763.743,E2 -27763.743} C_VEL
LIN {X 0,Y 103.001,Z 756.463,A -85,B 0,C 180,E1 -27765.01,E2 -27765.01} C_VEL
LIN {X 0,Y 94.261,Z 750.332,A -85,B 0,C 180,E1 -27773.382,E2 -27773.382} C_VEL
LIN {X 0,Y 89.238,Z 743.962,A -85,B 0,C 180,E1 -27781.801,E2 -27781.801} C_VEL
LIN {X 0,Y 86.891,Z 736.331,A -85,B 0,C 180,E1 -27791.123,E2 -27791.123} C_VEL
LIN {X 0,Y 86.766,Z 729.696,A -85,B 0,C 180,E1 -27798.08,E2 -27798.08} C_VEL
LIN {X 0,Y 88.096,Z 721.232,A -85,B 0,C 180,E1 -27805.425,E2 -27805.425} C_VEL
LIN {X 0,Y 88.473,Z 720.455,A -85,B 0,C 180,E1 -27806.277,E2 -27806.277} C_VEL
LIN {X 0,Y 85.947,Z 725.289,A -85,B 0,C 180,E1 -27810.873,E2 -27810.873} C_VEL
LIN {X 0,Y 84.689,Z 734.185,A -85,B 0,C 180,E1 -27819.554,E2 -27819.554} C_VEL
LIN {X 0,Y 84.798,Z 740.049,A -85,B 0,C 180,E1 -27826.863,E2 -27826.863} C_VEL
LIN {X 0,Y 86.81,Z 746.351,A -85,B 0,C 180,E1 -27835.989,E2 -27835.989} C_VEL
LIN {X 0,Y 93.208,Z 753.333,A -85,B 0,C 180,E1 -27847.101,E2 -27847.101} C_VEL
LIN {X 0,Y 100.624,Z 757.688,A -85,B 0,C 180,E1 -27854.303,E2 -27854.303} C_VEL
LIN {X 0,Y 103.746,Z 759.009,A -85,B 0,C 180,E1 -27857.357,E2 -27857.357} C_VEL
LIN {X 0,Y 94.481,Z 752.53,A -85,B 0,C 180,E1 -27864.91,E2 -27864.91} C_VEL
LIN {X 0,Y 87.833,Z 744.676,A -85,B 0,C 180,E1 -27873.891,E2 -27873.891} C_VEL
LIN {X 0,Y 84.562,Z 737.299,A -85,B 0,C 180,E1 -27881.84,E2 -27881.84} C_VEL
LIN {X 0,Y 83.062,Z 728.582,A -85,B 0,C 180,E1 -27890.257,E2 -27890.257} C_VEL
LIN {X 0,Y 82.458,Z 720.75,A -85,B 0,C 180,E1 -27896.335,E2 -27896.335} C_VEL
LIN {X 0,Y 82.118,Z 710.142,A -85,B 0,C 180,E1 -27903.066,E2 -27903.066} C_VEL
LIN {X 0,Y 82.211,Z 700.88,A -85,B 0,C 180,E1 -27907.985,E2 -27907.985} C_VEL
LIN {X 0,Y 83.016,Z 686.598,A -85,B 0,C 180,E1 -27914.087,E2 -27914.087} C_VEL
LIN {X 0,Y 84.114,Z 673.072,A -85,B 0,C 180,E1 -27918.575,E2 -27918.575} C_VEL
LIN {X 0,Y 84.366,Z 669.383,A -85,B 0,C 180,E1 -27919.614,E2 -27919.614} C_VEL
LIN {X 0,Y 84.03,Z 663.839,A -85,B 0,C 180,E1 -27920.927,E2 -27920.927} C_VEL
LIN {X 0,Y 79.641,Z 644.958,A -85,B 0,C 180,E1 -27924.187,E2 -27924.187} C_VEL
LIN {X 0,Y 79.458,Z 639.225,A -85,B 0,C 180,E1 -27925.256,E2 -27925.256} C_VEL
LIN {X 0,Y 83.413,Z 587.677,A -85,B 0,C 180,E1 -27934.886,E2 -27934.886} C_VEL
LIN {X 0,Y 81.987,Z 566.025,A -85,B 0,C 180,E1 -27938.782,E2 -27938.782} C_VEL
LIN {X 0,Y 74.466,Z 535.707,A -85,B 0,C 180,E1 -27945.416,E2 -27945.416} C_VEL
LIN {X 0,Y 72.891,Z 528.621,A -85,B 0,C 180,E1 -27953.261,E2 -27953.261} C_VEL
LIN {X 0,Y 72.453,Z 526.576,A -85,B 0,C 180,E1 -27955.681,E2 -27955.681} C_VEL
LIN {X 0,Y 72.393,Z 526.592,A -85,B 0,C 180,E1 -27960.96,E2 -27960.96} C_VEL
LIN {X 0,Y 72.4,Z 526.59,A -85,B 0,C 180,E1 -27967.152,E2 -27967.152} C_VEL
LIN {X 0,Y 72.758,Z 526.544,A -85,B 0,C 180,E1 -27975.002,E2 -27975.002} C_VEL
LIN {X 0,Y 72.886,Z 526.528,A -85,B 0,C 180,E1 -27978.88,E2 -27978.88} C_VEL
LIN {X 0,Y 73.582,Z 526.436,A -85,B 0,C 180,E1 -27990,E2 -27990} C_VEL
LIN {X 0,Y 72.886,Z 526.53,A -85,B 0,C 180,E1 -28001.119,E2 -28001.119} C_VEL
LIN {X 0,Y 72.587,Z 526.559,A -85,B 0,C 180,E1 -28006.885,E2 -28006.885} C_VEL
LIN {X 0,Y 72.401,Z 526.589,A -85,B 0,C 180,E1 -28012.847,E2 -28012.847} C_VEL
LIN {X 0,Y 72.377,Z 526.594,A -85,B 0,C 180,E1 -28019.082,E2 -28019.082} C_VEL
LIN {X 0,Y 72.44,Z 526.585,A -85,B 0,C 180,E1 -28029.508,E2 -28029.508} C_VEL
LIN {X 0,Y 72.478,Z 526.703,A -85,B 0,C 180,E1 -28030.05,E2 -28030.05} C_VEL
LIN {X 0,Y 75.137,Z 538.079,A -85,B 0,C 180,E1 -28037.442,E2 -28037.442} C_VEL
LIN {X 0,Y 78.13,Z 550.881,A -85,B 0,C 180,E1 -28045.135,E2 -28045.135} C_VEL
LIN {X 0,Y 78.858,Z 554.742,A -85,B 0,C 180,E1 -28047.21,E2 -28047.21} C_VEL
LIN {X 0,Y 80.077,Z 581.361,A -85,B 0,C 180,E1 -28051.95,E2 -28051.95} C_VEL
LIN {X 0,Y 80.6,Z 590.309,A -85,B 0,C 180,E1 -28053.523,E2 -28053.523} C_VEL
LIN {X 0,Y 78.53,Z 656.222,A -85,B 0,C 180,E1 -28066.578,E2 -28066.578} C_VEL
LIN {X 0,Y 78.139,Z 672.366,A -85,B 0,C 180,E1 -28070.357,E2 -28070.357} C_VEL
LIN {X 0,Y 77.759,Z 686.249,A -85,B 0,C 180,E1 -28074.815,E2 -28074.815} C_VEL
LIN {X 0,Y 77.757,Z 698.691,A -85,B 0,C 180,E1 -28080,E2 -28080} C_VEL
LIN {X 0,Y 78.223,Z 709.787,A -85,B 0,C 180,E1 -28085.801,E2 -28085.801} C_VEL
LIN {X 0,Y 78.933,Z 718.047,A -85,B 0,C 180,E1 -28091.12,E2 -28091.12} C_VEL
LIN {X 0,Y 79.624,Z 725.028,A -85,B 0,C 180,E1 -28096.67,E2 -28096.67} C_VEL
LIN {X 0,Y 82.373,Z 735.421,A -85,B 0,C 180,E1 -28106.611,E2 -28106.611} C_VEL
LIN {X 0,Y 87.414,Z 743.748,A -85,B 0,C 180,E1 -28115.311,E2 -28115.311} C_VEL
LIN {X 0,Y 94.024,Z 750.352,A -85,B 0,C 180,E1 -28122.278,E2 -28122.278} C_VEL
LIN {X 0,Y 95.906,Z 751.812,A -85,B 0,C 180,E1 -28123.82,E2 -28123.82} C_VEL
LIN {X 0,Y 94.679,Z 751.097,A -85,B 0,C 180,E1 -28125.459,E2 -28125.459} C_VEL
LIN {X 0,Y 86.325,Z 743.714,A -85,B 0,C 180,E1 -28135.258,E2 -28135.258} C_VEL
LIN {X 0,Y 82.028,Z 735.407,A -85,B 0,C 180,E1 -28145.986,E2 -28145.986} C_VEL
LIN {X 0,Y 81.161,Z 727.525,A -85,B 0,C 180,E1 -28154.943,E2 -28154.943} C_VEL
LIN {X 0,Y 81.994,Z 718.774,A -85,B 0,C 180,E1 -28163.01,E2 -28163.01} C_VEL
LIN {X 0,Y 83.108,Z 715.837,A -85,B 0,C 180,E1 -28165.909,E2 -28165.909} C_VEL
LIN {X 0,Y 80.582,Z 719.986,A -85,B 0,C 180,E1 -28170,E2 -28170} C_VEL
LIN {X 0,Y 78.847,Z 727.687,A -85,B 0,C 180,E1 -28177.684,E2 -28177.684} C_VEL
LIN {X 0,Y 78.803,Z 733.306,A -85,B 0,C 180,E1 -28184.066,E2 -28184.066} C_VEL
LIN {X 0,Y 79.87,Z 739.942,A -85,B 0,C 180,E1 -28193.327,E2 -28193.327} C_VEL
LIN {X 0,Y 85.017,Z 747.677,A -85,B 0,C 180,E1 -28205.357,E2 -28205.357} C_VEL
LIN {X 0,Y 94.818,Z 754.367,A -85,B 0,C 180,E1 -28216.077,E2 -28216.077} C_VEL
LIN {X 0,Y 94.326,Z 753.865,A -85,B 0,C 180,E1 -28217.889,E2 -28217.889} C_VEL
LIN {X 0,Y 86.581,Z 747.333,A -85,B 0,C 180,E1 -28225.375,E2 -28225.375} C_VEL
LIN {X 0,Y 80.384,Z 738.405,A -85,B 0,C 180,E1 -28235.462,E2 -28235.462} C_VEL
LIN {X 0,Y 77.734,Z 730.095,A -85,B 0,C 180,E1 -28244.262,E2 -28244.262} C_VEL
LIN {X 0,Y 76.761,Z 723.008,A -85,B 0,C 180,E1 -28250.78,E2 -28250.78} C_VEL
LIN {X 0,Y 76.138,Z 716.239,A -85,B 0,C 180,E1 -28256.03,E2 -28256.03} C_VEL
LIN {X 0,Y 75.671,Z 705.804,A -85,B 0,C 180,E1 -28262.662,E2 -28262.662} C_VEL
LIN {X 0,Y 75.711,Z 695.799,A -85,B 0,C 180,E1 -28268.004,E2 -28268.004} C_VEL
LIN {X 0,Y 76.494,Z 682.311,A -85,B 0,C 180,E1 -28273.956,E2 -28273.956} C_VEL
LIN {X 0,Y 77.416,Z 670.042,A -85,B 0,C 180,E1 -28278.184,E2 -28278.184} C_VEL
LIN {X 0,Y 78.529,Z 653.592,A -85,B 0,C 180,E1 -28282.356,E2 -28282.356} C_VEL
LIN {X 0,Y 79.458,Z 639.225,A -85,B 0,C 180,E1 -28285.256,E2 -28285.256} C_VEL
LIN {X 0,Y 79.305,Z 633.528,A -85,B 0,C 180,E1 -28286.335,E2 -28286.335} C_VEL
LIN {X 0,Y 77.175,Z 624.135,A -85,B 0,C 180,E1 -28287.996,E2 -28287.996} C_VEL
LIN {X 0,Y 74.867,Z 614.725,A -85,B 0,C 180,E1 -28289.724,E2 -28289.724} C_VEL
LIN {X 0,Y 74.482,Z 608.99,A -85,B 0,C 180,E1 -28290.856,E2 -28290.856} C_VEL
LIN {X 0,Y 76.327,Z 587.92,A -85,B 0,C 180,E1 -28295.02,E2 -28295.02} C_VEL
LIN {X 0,Y 74.998,Z 567.299,A -85,B 0,C 180,E1 -28299.088,E2 -28299.088} C_VEL
LIN {X 0,Y 68.188,Z 539.62,A -85,B 0,C 180,E1 -28305.608,E2 -28305.608} C_VEL
LIN {X 0,Y 67.211,Z 535.648,A -85,B 0,C 180,E1 -28306.663,E2 -28306.663} C_VEL
LIN {X 0,Y 65.561,Z 528.288,A -85,B 0,C 180,E1 -28315.751,E2 -28315.751} C_VEL
LIN {X 0,Y 65.334,Z 527.465,A -85,B 0,C 180,E1 -28317.004,E2 -28317.004} C_VEL
LIN {X 0,Y 65.249,Z 527.473,A -85,B 0,C 180,E1 -28324.478,E2 -28324.478} C_VEL
LIN {X 0,Y 65.652,Z 527.427,A -85,B 0,C 180,E1 -28334.459,E2 -28334.459} C_VEL
LIN {X 0,Y 65.784,Z 527.415,A -85,B 0,C 180,E1 -28337.662,E2 -28337.662} C_VEL
LIN {X 0,Y 66.506,Z 527.317,A -85,B 0,C 180,E1 -28350,E2 -28350} C_VEL
LIN {X 0,Y 65.784,Z 527.416,A -85,B 0,C 180,E1 -28362.337,E2 -28362.337} C_VEL
LIN {X 0,Y 65.392,Z 527.461,A -85,B 0,C 180,E1 -28368.809,E2 -28368.809} C_VEL
LIN {X 0,Y 65.249,Z 527.474,A -85,B 0,C 180,E1 -28375.521,E2 -28375.521} C_VEL
LIN {X 0,Y 65.211,Z 527.48,A -85,B 0,C 180,E1 -28382.606,E2 -28382.606} C_VEL
LIN {X 0,Y 65.428,Z 527.583,A -85,B 0,C 180,E1 -28389.129,E2 -28389.129} C_VEL
LIN {X 0,Y 67.806,Z 537.902,A -85,B 0,C 180,E1 -28396.514,E2 -28396.514} C_VEL
LIN {X 0,Y 70.85,Z 550.766,A -85,B 0,C 180,E1 -28404.921,E2 -28404.921} C_VEL
LIN {X 0,Y 71.777,Z 555.142,A -85,B 0,C 180,E1 -28407.42,E2 -28407.42} C_VEL
LIN {X 0,Y 73.149,Z 583.239,A -85,B 0,C 180,E1 -28412.847,E2 -28412.847} C_VEL
LIN {X 0,Y 73.566,Z 590.065,A -85,B 0,C 180,E1 -28414.159,E2 -28414.159} C_VEL
LIN {X 0,Y 71.978,Z 655.349,A -85,B 0,C 180,E1 -28428.561,E2 -28428.561} C_VEL
LIN {X 0,Y 71.752,Z 671.394,A -85,B 0,C 180,E1 -28432.614,E2 -28432.614} C_VEL
LIN {X 0,Y 71.593,Z 684.658,A -85,B 0,C 180,E1 -28437.187,E2 -28437.187} C_VEL
LIN {X 0,Y 71.844,Z 696.818,A -85,B 0,C 180,E1 -28442.628,E2 -28442.628} C_VEL
LIN {X 0,Y 72.588,Z 707.754,A -85,B 0,C 180,E1 -28448.701,E2 -28448.701} C_VEL
LIN {X 0,Y 73.433,Z 715.431,A -85,B 0,C 180,E1 -28453.843,E2 -28453.843} C_VEL
LIN {X 0,Y 74.282,Z 721.436,A -85,B 0,C 180,E1 -28458.892,E2 -28458.892} C_VEL
LIN {X 0,Y 77.084,Z 731.39,A -85,B 0,C 180,E1 -28468.598,E2 -28468.598} C_VEL
LIN {X 0,Y 82.792,Z 740.611,A -85,B 0,C 180,E1 -28478.254,E2 -28478.254} C_VEL
LIN {X 0,Y 88.524,Z 746.375,A -85,B 0,C 180,E1 -28484.397,E2 -28484.397} C_VEL
LIN {X 0,Y 81.508,Z 739.848,A -85,B 0,C 180,E1 -28492.874,E2 -28492.874} C_VEL
LIN {X 0,Y 77.186,Z 732.187,A -85,B 0,C 180,E1 -28502.918,E2 -28502.918} C_VEL
LIN {X 0,Y 75.843,Z 724.228,A -85,B 0,C 180,E1 -28512.419,E2 -28512.419} C_VEL
LIN {X 0,Y 76.6,Z 714.263,A -85,B 0,C 180,E1 -28522.093,E2 -28522.093} C_VEL
LIN {X 0,Y 77.996,Z 710.965,A -85,B 0,C 180,E1 -28525.413,E2 -28525.413} C_VEL
LIN {X 0,Y 75.041,Z 715.418,A -85,B 0,C 180,E1 -28530,E2 -28530} C_VEL
LIN {X 0,Y 73.101,Z 723.274,A -85,B 0,C 180,E1 -28538.292,E2 -28538.292} C_VEL
LIN {X 0,Y 73.071,Z 728.245,A -85,B 0,C 180,E1 -28543.916,E2 -28543.916} C_VEL
LIN {X 0,Y 73.78,Z 734.278,A -85,B 0,C 180,E1 -28552.398,E2 -28552.398} C_VEL
LIN {X 0,Y 77.19,Z 741.184,A -85,B 0,C 180,E1 -28563.113,E2 -28563.113} C_VEL
LIN {X 0,Y 85.343,Z 748.363,A -85,B 0,C 180,E1 -28574.426,E2 -28574.426} C_VEL
LIN {X 0,Y 87.366,Z 749.62,A -85,B 0,C 180,E1 -28576.386,E2 -28576.386} C_VEL
LIN {X 0,Y 83.243,Z 746.054,A -85,B 0,C 180,E1 -28580.713,E2 -28580.713} C_VEL
LIN {X 0,Y 76.596,Z 738.179,A -85,B 0,C 180,E1 -28589.692,E2 -28589.692} C_VEL
LIN {X 0,Y 72.133,Z 727.53,A -85,B 0,C 180,E1 -28601.539,E2 -28601.539} C_VEL
LIN {X 0,Y 70.907,Z 720.198,A -85,B 0,C 180,E1 -28608.566,E2 -28608.566} C_VEL
LIN {X 0,Y 70.058,Z 713.14,A -85,B 0,C 180,E1 -28614.242,E2 -28614.242} C_VEL
LIN {X 0,Y 69.394,Z 703.622,A -85,B 0,C 180,E1 -28620.725,E2 -28620.725} C_VEL
LIN {X 0,Y 69.269,Z 693.265,A -85,B 0,C 180,E1 -28626.554,E2 -28626.554} C_VEL
LIN {X 0,Y 69.836,Z 681.001,A -85,B 0,C 180,E1 -28632.348,E2 -28632.348} C_VEL
LIN {X 0,Y 70.69,Z 667.412,A -85,B 0,C 180,E1 -28637.353,E2 -28637.353} C_VEL
LIN {X 0,Y 71.662,Z 652.086,A -85,B 0,C 180,E1 -28641.578,E2 -28641.578} C_VEL
LIN {X 0,Y 74.482,Z 608.99,A -85,B 0,C 180,E1 -28650.856,E2 -28650.856} C_VEL
LIN {X 0,Y 74.115,Z 603.244,A -85,B 0,C 180,E1 -28652.007,E2 -28652.007} C_VEL
LIN {X 0,Y 68.903,Z 582.572,A -85,B 0,C 180,E1 -28656.366,E2 -28656.366} C_VEL
LIN {X 0,Y 68.602,Z 578.719,A -85,B 0,C 180,E1 -28657.196,E2 -28657.196} C_VEL
LIN {X 0,Y 67.982,Z 568.404,A -85,B 0,C 180,E1 -28659.45,E2 -28659.45} C_VEL
LIN {X 0,Y 60.986,Z 539.767,A -85,B 0,C 180,E1 -28666.824,E2 -28666.824} C_VEL
LIN {X 0,Y 59.91,Z 535.524,A -85,B 0,C 180,E1 -28668.148,E2 -28668.148} C_VEL
LIN {X 0,Y 58.367,Z 528.853,A -85,B 0,C 180,E1 -28677.444,E2 -28677.444} C_VEL
LIN {X 0,Y 58.269,Z 528.349,A -85,B 0,C 180,E1 -28678.223,E2 -28678.223} C_VEL
LIN {X 0,Y 58.197,Z 528.361,A -85,B 0,C 180,E1 -28688.759,E2 -28688.759} C_VEL
LIN {X 0,Y 58.66,Z 528.303,A -85,B 0,C 180,E1 -28696.135,E2 -28696.135} C_VEL
LIN {X 0,Y 58.827,Z 528.277,A -85,B 0,C 180,E1 -28703.138,E2 -28703.138} C_VEL
LIN {X 0,Y 59.399,Z 528.202,A -85,B 0,C 180,E1 -28710,E2 -28710} C_VEL
LIN {X 0,Y 58.826,Z 528.275,A -85,B 0,C 180,E1 -28716.861,E2 -28716.861} C_VEL
LIN {X 0,Y 58.538,Z 528.309,A -85,B 0,C 180,E1 -28726.165,E2 -28726.165} C_VEL
LIN {X 0,Y 58.157,Z 528.365,A -85,B 0,C 180,E1 -28738.906,E2 -28738.906} C_VEL
LIN {X 0,Y 58.323,Z 528.486,A -85,B 0,C 180,E1 -28748.139,E2 -28748.139} C_VEL
LIN {X 0,Y 60.624,Z 538.328,A -85,B 0,C 180,E1 -28755.928,E2 -28755.928} C_VEL
LIN {X 0,Y 63.698,Z 550.999,A -85,B 0,C 180,E1 -28765.01,E2 -28765.01} C_VEL
LIN {X 0,Y 64.629,Z 554.783,A -85,B 0,C 180,E1 -28767.554,E2 -28767.554} C_VEL
LIN {X 0,Y 66.341,Z 585.683,A -85,B 0,C 180,E1 -28774.232,E2 -28774.232} C_VEL
LIN {X 0,Y 66.541,Z 590.226,A -85,B 0,C 180,E1 -28775.218,E2 -28775.218} C_VEL
LIN {X 0,Y 65.55,Z 654.568,A -85,B 0,C 180,E1 -28790.988,E2 -28790.988} C_VEL
LIN {X 0,Y 65.586,Z 670.291,A -85,B 0,C 180,E1 -28795.39,E2 -28795.39} C_VEL
LIN {X 0,Y 65.703,Z 684.439,A -85,B 0,C 180,E1 -28800.766,E2 -28800.766} C_VEL
LIN {X 0,Y 66.208,Z 695.473,A -85,B 0,C 180,E1 -28806.094,E2 -28806.094} C_VEL
LIN {X 0,Y 67.222,Z 705.604,A -85,B 0,C 180,E1 -28812.07,E2 -28812.07} C_VEL
LIN {X 0,Y 68.462,Z 713.667,A -85,B 0,C 180,E1 -28817.937,E2 -28817.937} C_VEL
LIN {X 0,Y 69.635,Z 720.154,A -85,B 0,C 180,E1 -28823.81,E2 -28823.81} C_VEL
LIN {X 0,Y 73.965,Z 730.81,A -85,B 0,C 180,E1 -28834.758,E2 -28834.758} C_VEL
LIN {X 0,Y 80.876,Z 739.705,A -85,B 0,C 180,E1 -28844.042,E2 -28844.042} C_VEL
LIN {X 0,Y 80.376,Z 739.326,A -85,B 0,C 180,E1 -28845.612,E2 -28845.612} C_VEL
LIN {X 0,Y 73.105,Z 729.922,A -85,B 0,C 180,E1 -28858.079,E2 -28858.079} C_VEL
LIN {X 0,Y 70.791,Z 720.958,A -85,B 0,C 180,E1 -28869.342,E2 -28869.342} C_VEL
LIN {X 0,Y 71.282,Z 710.137,A -85,B 0,C 180,E1 -28880.384,E2 -28880.384} C_VEL
LIN {X 0,Y 73.079,Z 705.924,A -85,B 0,C 180,E1 -28884.828,E2 -28884.828} C_VEL
LIN {X 0,Y 69.725,Z 710.531,A -85,B 0,C 180,E1 -28890,E2 -28890} C_VEL
LIN {X 0,Y 67.538,Z 718.284,A -85,B 0,C 180,E1 -28898.58,E2 -28898.58} C_VEL
LIN {X 0,Y 67.597,Z 725.011,A -85,B 0,C 180,E1 -28906.616,E2 -28906.616} C_VEL
LIN {X 0,Y 70.016,Z 734.007,A -85,B 0,C 180,E1 -28920.125,E2 -28920.125} C_VEL
LIN {X 0,Y 77.193,Z 742.168,A -85,B 0,C 180,E1 -28933.251,E2 -28933.251} C_VEL
LIN {X 0,Y 78.971,Z 743.566,A -85,B 0,C 180,E1 -28935.395,E2 -28935.395} C_VEL
LIN {X 0,Y 78.203,Z 742.631,A -85,B 0,C 180,E1 -28938.003,E2 -28938.003} C_VEL
LIN {X 0,Y 70.582,Z 733.419,A -85,B 0,C 180,E1 -28948.483,E2 -28948.483} C_VEL
LIN {X 0,Y 66.463,Z 723.3,A -85,B 0,C 180,E1 -28959.9,E2 -28959.9} C_VEL
LIN {X 0,Y 65.244,Z 717.461,A -85,B 0,C 180,E1 -28965.81,E2 -28965.81} C_VEL
LIN {X 0,Y 64.006,Z 708.843,A -85,B 0,C 180,E1 -28972.904,E2 -28972.904} C_VEL
LIN {X 0,Y 63.144,Z 697.42,A -85,B 0,C 180,E1 -28980.797,E2 -28980.797} C_VEL
LIN {X 0,Y 63.14,Z 683.001,A -85,B 0,C 180,E1 -28988.804,E2 -28988.804} C_VEL
LIN {X 0,Y 63.804,Z 669.081,A -85,B 0,C 180,E1 -28994.757,E2 -28994.757} C_VEL
LIN {X 0,Y 64.655,Z 652.806,A -85,B 0,C 180,E1 -28999.858,E2 -28999.858} C_VEL
LIN {X 0,Y 67.409,Z 608.548,A -85,B 0,C 180,E1 -29010.625,E2 -29010.625} C_VEL
LIN {X 0,Y 69.195,Z 587.538,A -85,B 0,C 180,E1 -29015.303,E2 -29015.303} C_VEL
LIN {X 0,Y 68.602,Z 578.719,A -85,B 0,C 180,E1 -29017.196,E2 -29017.196} C_VEL
LIN {X 0,Y 68.121,Z 574.962,A -85,B 0,C 180,E1 -29018.022,E2 -29018.022} C_VEL
LIN {X 0,Y 66.087,Z 569.61,A -85,B 0,C 180,E1 -29019.303,E2 -29019.303} C_VEL
LIN {X 0,Y 58.233,Z 556.147,A -85,B 0,C 180,E1 -29023.264,E2 -29023.264} C_VEL
LIN {X 0,Y 56.345,Z 550.657,A -85,B 0,C 180,E1 -29024.954,E2 -29024.954} C_VEL
LIN {X 0,Y 52.622,Z 535.385,A -85,B 0,C 180,E1 -29029.971,E2 -29029.971} C_VEL
LIN {X 0,Y 51.195,Z 529.233,A -85,B 0,C 180,E1 -29039.871,E2 -29039.871} C_VEL
LIN {X 0,Y 51.483,Z 529.189,A -85,B 0,C 180,E1 -29054.155,E2 -29054.155} C_VEL
LIN {X 0,Y 51.702,Z 529.161,A -85,B 0,C 180,E1 -29062.187,E2 -29062.187} C_VEL
LIN {X 0,Y 52.284,Z 529.088,A -85,B 0,C 180,E1 -29070,E2 -29070} C_VEL
LIN {X 0,Y 51.702,Z 529.16,A -85,B 0,C 180,E1 -29077.812,E2 -29077.812} C_VEL
LIN {X 0,Y 51.404,Z 529.197,A -85,B 0,C 180,E1 -29086.856,E2 -29086.856} C_VEL
LIN {X 0,Y 51.03,Z 529.245,A -85,B 0,C 180,E1 -29094.404,E2 -29094.404} C_VEL
LIN {X 0,Y 51.219,Z 529.228,A -85,B 0,C 180,E1 -29106.689,E2 -29106.689} C_VEL
LIN {X 0,Y 53.393,Z 538.446,A -85,B 0,C 180,E1 -29115.031,E2 -29115.031} C_VEL
LIN {X 0,Y 56.575,Z 551.361,A -85,B 0,C 180,E1 -29125.384,E2 -29125.384} C_VEL
LIN {X 0,Y 57.553,Z 555.188,A -85,B 0,C 180,E1 -29128.11,E2 -29128.11} C_VEL
LIN {X 0,Y 59.42,Z 586.301,A -85,B 0,C 180,E1 -29135.546,E2 -29135.546} C_VEL
LIN {X 0,Y 59.561,Z 590.329,A -85,B 0,C 180,E1 -29136.532,E2 -29136.532} C_VEL
LIN {X 0,Y 59.37,Z 653.631,A -85,B 0,C 180,E1 -29154.055,E2 -29154.055} C_VEL
LIN {X 0,Y 59.675,Z 670.134,A -85,B 0,C 180,E1 -29159.157,E2 -29159.157} C_VEL
LIN {X 0,Y 60.028,Z 682.449,A -85,B 0,C 180,E1 -29164.197,E2 -29164.197} C_VEL
LIN {X 0,Y 60.923,Z 693.55,A -85,B 0,C 180,E1 -29169.965,E2 -29169.965} C_VEL
LIN {X 0,Y 62.337,Z 703.745,A -85,B 0,C 180,E1 -29176.371,E2 -29176.371} C_VEL
LIN {X 0,Y 63.923,Z 712.02,A -85,B 0,C 180,E1 -29182.805,E2 -29182.805} C_VEL
LIN {X 0,Y 67.242,Z 722.403,A -85,B 0,C 180,E1 -29193.265,E2 -29193.265} C_VEL
LIN {X 0,Y 72.698,Z 731.186,A -85,B 0,C 180,E1 -29202.588,E2 -29202.588} C_VEL
LIN {X 0,Y 74.034,Z 732.913,A -85,B 0,C 180,E1 -29205.484,E2 -29205.484} C_VEL
LIN {X 0,Y 67.547,Z 723.045,A -85,B 0,C 180,E1 -29218.653,E2 -29218.653} C_VEL
LIN {X 0,Y 65.871,Z 715.383,A -85,B 0,C 180,E1 -29228.301,E2 -29228.301} C_VEL
LIN {X 0,Y 66.026,Z 706.512,A -85,B 0,C 180,E1 -29237.709,E2 -29237.709} C_VEL
LIN {X 0,Y 67.515,Z 702.1,A -85,B 0,C 180,E1 -29242.522,E2 -29242.522} C_VEL
LIN {X 0,Y 68.35,Z 700.67,A -85,B 0,C 180,E1 -29244.284,E2 -29244.284} C_VEL
LIN {X 0,Y 65.417,Z 704.129,A -85,B 0,C 180,E1 -29248.433,E2 -29248.433} C_VEL
LIN {X 0,Y 62.94,Z 709.446,A -85,B 0,C 180,E1 -29254.646,E2 -29254.646} C_VEL
LIN {X 0,Y 62.063,Z 718.103,A -85,B 0,C 180,E1 -29265.055,E2 -29265.055} C_VEL
LIN {X 0,Y 62.85,Z 724.125,A -85,B 0,C 180,E1 -29273.548,E2 -29273.548} C_VEL
LIN {X 0,Y 66.277,Z 731.626,A -85,B 0,C 180,E1 -29285.678,E2 -29285.678} C_VEL
LIN {X 0,Y 70.941,Z 736.738,A -85,B 0,C 180,E1 -29293.907,E2 -29293.907} C_VEL
LIN {X 0,Y 71.799,Z 737.302,A -85,B 0,C 180,E1 -29296.749,E2 -29296.749} C_VEL
LIN {X 0,Y 64.087,Z 727.039,A -85,B 0,C 180,E1 -29308.607,E2 -29308.607} C_VEL
LIN {X 0,Y 60.579,Z 717.319,A -85,B 0,C 180,E1 -29319.632,E2 -29319.632} C_VEL
LIN {X 0,Y 59.029,Z 710.409,A -85,B 0,C 180,E1 -29326.224,E2 -29326.224} C_VEL
LIN {X 0,Y 57.761,Z 702.029,A -85,B 0,C 180,E1 -29333.011,E2 -29333.011} C_VEL
LIN {X 0,Y 56.987,Z 693.19,A -85,B 0,C 180,E1 -29339.117,E2 -29339.117} C_VEL
LIN {X 0,Y 56.819,Z 679.612,A -85,B 0,C 180,E1 -29347.105,E2 -29347.105} C_VEL
LIN {X 0,Y 57.258,Z 666.446,A -85,B 0,C 180,E1 -29353.215,E2 -29353.215} C_VEL
LIN {X 0,Y 57.889,Z 651.44,A -85,B 0,C 180,E1 -29358.354,E2 -29358.354} C_VEL
LIN {X 0,Y 62.13,Z 588.935,A -85,B 0,C 180,E1 -29374.97,E2 -29374.97} C_VEL
LIN {X 0,Y 60.894,Z 569.377,A -85,B 0,C 180,E1 -29379.698,E2 -29379.698} C_VEL
LIN {X 0,Y 56.345,Z 550.657,A -85,B 0,C 180,E1 -29384.954,E2 -29384.954} C_VEL
LIN {X 0,Y 55.074,Z 546.924,A -85,B 0,C 180,E1 -29386.246,E2 -29386.246} C_VEL
LIN {X 0,Y 52.183,Z 542.515,A -85,B 0,C 180,E1 -29388.08,E2 -29388.08} C_VEL
LIN {X 0,Y 45.724,Z 535.544,A -85,B 0,C 180,E1 -29392.168,E2 -29392.168} C_VEL
LIN {X 0,Y 45.093,Z 534.333,A -85,B 0,C 180,E1 -29393.803,E2 -29393.803} C_VEL
LIN {X 0,Y 44.047,Z 530.117,A -85,B 0,C 180,E1 -29402.049,E2 -29402.049} C_VEL
LIN {X 0,Y 44.259,Z 530.087,A -85,B 0,C 180,E1 -29412.317,E2 -29412.317} C_VEL
LIN {X 0,Y 44.554,Z 530.051,A -85,B 0,C 180,E1 -29420.924,E2 -29420.924} C_VEL
LIN {X 0,Y 45.159,Z 529.975,A -85,B 0,C 180,E1 -29429.999,E2 -29429.999} C_VEL
LIN {X 0,Y 44.553,Z 530.051,A -85,B 0,C 180,E1 -29439.075,E2 -29439.075} C_VEL
LIN {X 0,Y 44.195,Z 530.098,A -85,B 0,C 180,E1 -29448.544,E2 -29448.544} C_VEL
LIN {X 0,Y 44.118,Z 530.173,A -85,B 0,C 180,E1 -29465.47,E2 -29465.47} C_VEL
LIN {X 0,Y 46.001,Z 537.908,A -85,B 0,C 180,E1 -29473.432,E2 -29473.432} C_VEL
LIN {X 0,Y 49.596,Z 552.166,A -85,B 0,C 180,E1 -29486.346,E2 -29486.346} C_VEL
LIN {X 0,Y 50.399,Z 555.23,A -85,B 0,C 180,E1 -29488.777,E2 -29488.777} C_VEL
LIN {X 0,Y 52.695,Z 589.783,A -85,B 0,C 180,E1 -29498.227,E2 -29498.227} C_VEL
LIN {X 0,Y 53.412,Z 652.792,A -85,B 0,C 180,E1 -29517.879,E2 -29517.879} C_VEL
LIN {X 0,Y 54.094,Z 669.019,A -85,B 0,C 180,E1 -29523.492,E2 -29523.492} C_VEL
LIN {X 0,Y 54.878,Z 681.769,A -85,B 0,C 180,E1 -29529.212,E2 -29529.212} C_VEL
LIN {X 0,Y 56.22,Z 692.891,A -85,B 0,C 180,E1 -29535.405,E2 -29535.405} C_VEL
LIN {X 0,Y 58.134,Z 702.87,A -85,B 0,C 180,E1 -29542.193,E2 -29542.193} C_VEL
LIN {X 0,Y 59.915,Z 709.697,A -85,B 0,C 180,E1 -29547.983,E2 -29547.983} C_VEL
LIN {X 0,Y 63.466,Z 718.891,A -85,B 0,C 180,E1 -29557.521,E2 -29557.521} C_VEL
LIN {X 0,Y 67.905,Z 725.778,A -85,B 0,C 180,E1 -29564.848,E2 -29564.848} C_VEL
LIN {X 0,Y 66.864,Z 724.55,A -85,B 0,C 180,E1 -29567.372,E2 -29567.372} C_VEL
LIN {X 0,Y 62.041,Z 714.744,A -85,B 0,C 180,E1 -29580.689,E2 -29580.689} C_VEL
LIN {X 0,Y 60.937,Z 707.142,A -85,B 0,C 180,E1 -29589.758,E2 -29589.758} C_VEL
LIN {X 0,Y 61.4,Z 700.844,A -85,B 0,C 180,E1 -29596.767,E2 -29596.767} C_VEL
LIN {X 0,Y 63.704,Z 695.458,A -85,B 0,C 180,E1 -29603.171,E2 -29603.171} C_VEL
LIN {X 0,Y 63.906,Z 695.183,A -85,B 0,C 180,E1 -29603.687,E2 -29603.687} C_VEL
LIN {X 0,Y 60.56,Z 698.807,A -85,B 0,C 180,E1 -29608.307,E2 -29608.307} C_VEL
LIN {X 0,Y 57.364,Z 705.789,A -85,B 0,C 180,E1 -29617.038,E2 -29617.038} C_VEL
LIN {X 0,Y 57.322,Z 716.815,A -85,B 0,C 180,E1 -29631.582,E2 -29631.582} C_VEL
LIN {X 0,Y 59.327,Z 723.41,A -85,B 0,C 180,E1 -29642.214,E2 -29642.214} C_VEL
LIN {X 0,Y 64.975,Z 730.909,A -85,B 0,C 180,E1 -29654.674,E2 -29654.674} C_VEL
LIN {X 0,Y 64.312,Z 729.987,A -85,B 0,C 180,E1 -29657.048,E2 -29657.048} C_VEL
LIN {X 0,Y 57.201,Z 718.582,A -85,B 0,C 180,E1 -29670.563,E2 -29670.563} C_VEL
LIN {X 0,Y 55.154,Z 712.372,A -85,B 0,C 180,E1 -29677.525,E2 -29677.525} C_VEL
LIN {X 0,Y 53.261,Z 704.76,A -85,B 0,C 180,E1 -29684.698,E2 -29684.698} C_VEL
LIN {X 0,Y 51.544,Z 694.334,A -85,B 0,C 180,E1 -29693.148,E2 -29693.148} C_VEL
LIN {X 0,Y 50.637,Z 680.281,A -85,B 0,C 180,E1 -29702.486,E2 -29702.486} C_VEL
LIN {X 0,Y 50.784,Z 666.17,A -85,B 0,C 180,E1 -29709.961,E2 -29709.961} C_VEL
LIN {X 0,Y 51.254,Z 649.894,A -85,B 0,C 180,E1 -29716.289,E2 -29716.289} C_VEL
LIN {X 0,Y 55.029,Z 588.358,A -85,B 0,C 180,E1 -29735.08,E2 -29735.08} C_VEL
LIN {X 0,Y 53.891,Z 570.425,A -85,B 0,C 180,E1 -29739.989,E2 -29739.989} C_VEL
LIN {X 0,Y 47.2,Z 542.549,A -85,B 0,C 180,E1 -29749.167,E2 -29749.167} C_VEL
LIN {X 0,Y 45.286,Z 535.148,A -85,B 0,C 180,E1 -29752.332,E2 -29752.332} C_VEL
LIN {X 0,Y 45.093,Z 534.333,A -85,B 0,C 180,E1 -29753.803,E2 -29753.803} C_VEL
LIN {X 0,Y 44.266,Z 532.771,A -85,B 0,C 180,E1 -29757.295,E2 -29757.295} C_VEL
LIN {X 0,Y 42.184,Z 531.492,A -85,B 0,C 180,E1 -29762.51,E2 -29762.51} C_VEL
LIN {X 0,Y 37.922,Z 530.932,A -85,B 0,C 180,E1 -29775.015,E2 -29775.015} C_VEL
LIN {X 0,Y 37.376,Z 530.933,A -85,B 0,C 180,E1 -29781.354,E2 -29781.354} C_VEL
LIN {X 0,Y 38.018,Z 530.864,A -85,B 0,C 180,E1 -29789.999,E2 -29789.999} C_VEL
LIN {X 0,Y 37.351,Z 530.952,A -85,B 0,C 180,E1 -29800.845,E2 -29800.845} C_VEL
LIN {X 0,Y 37.084,Z 530.983,A -85,B 0,C 180,E1 -29808.634,E2 -29808.634} C_VEL
LIN {X 0,Y 37.022,Z 530.988,A -85,B 0,C 180,E1 -29823.483,E2 -29823.483} C_VEL
LIN {X 0,Y 38.859,Z 538.343,A -85,B 0,C 180,E1 -29832.551,E2 -29832.551} C_VEL
LIN {X 0,Y 42.557,Z 552.725,A -85,B 0,C 180,E1 -29847.527,E2 -29847.527} C_VEL
LIN {X 0,Y 43.387,Z 555.819,A -85,B 0,C 180,E1 -29850.111,E2 -29850.111} C_VEL
LIN {X 0,Y 45.874,Z 589.22,A -85,B 0,C 180,E1 -29860.477,E2 -29860.477} C_VEL
LIN {X 0,Y 47.903,Z 652.114,A -85,B 0,C 180,E1 -29882.891,E2 -29882.891} C_VEL
LIN {X 0,Y 48.989,Z 667.742,A -85,B 0,C 180,E1 -29888.768,E2 -29888.768} C_VEL
LIN {X 0,Y 50.284,Z 681.092,A -85,B 0,C 180,E1 -29895.193,E2 -29895.193} C_VEL
LIN {X 0,Y 52.173,Z 691.969,A -85,B 0,C 180,E1 -29901.743,E2 -29901.743} C_VEL
LIN {X 0,Y 54.364,Z 700.64,A -85,B 0,C 180,E1 -29907.945,E2 -29907.945} C_VEL
LIN {X 0,Y 56.421,Z 707.225,A -85,B 0,C 180,E1 -29913.836,E2 -29913.836} C_VEL
LIN {X 0,Y 61.046,Z 716.549,A -85,B 0,C 180,E1 -29923.691,E2 -29923.691} C_VEL
LIN {X 0,Y 61.703,Z 717.604,A -85,B 0,C 180,E1 -29926.89,E2 -29926.89} C_VEL
LIN {X 0,Y 57.33,Z 707.545,A -85,B 0,C 180,E1 -29940.636,E2 -29940.636} C_VEL
LIN {X 0,Y 56.816,Z 696.146,A -85,B 0,C 180,E1 -29954.155,E2 -29954.155} C_VEL
LIN {X 0,Y 59.01,Z 690.478,A -85,B 0,C 180,E1 -29961.437,E2 -29961.437} C_VEL
LIN {X 0,Y 59.744,Z 689.49,A -85,B 0,C 180,E1 -29962.98,E2 -29962.98} C_VEL
LIN {X 0,Y 56.276,Z 692.81,A -85,B 0,C 180,E1 -29967.542,E2 -29967.542} C_VEL
LIN {X 0,Y 52.803,Z 699.187,A -85,B 0,C 180,E1 -29976.141,E2 -29976.141} C_VEL
LIN {X 0,Y 51.908,Z 709.022,A -85,B 0,C 180,E1 -29989.781,E2 -29989.781} C_VEL
LIN {X 0,Y 53.001,Z 714.171,A -85,B 0,C 180,E1 -29997.445,E2 -29997.445} C_VEL
LIN {X 0,Y 58.345,Z 723.68,A -85,B 0,C 180,E1 -30013.718,E2 -30013.718} C_VEL
LIN {X 0,Y 57.207,Z 722.032,A -85,B 0,C 180,E1 -30017.487,E2 -30017.487} C_VEL
LIN {X 0,Y 51.752,Z 712.239,A -85,B 0,C 180,E1 -30029.277,E2 -30029.277} C_VEL
LIN {X 0,Y 49.854,Z 707.02,A -85,B 0,C 180,E1 -30034.981,E2 -30034.981} C_VEL
LIN {X 0,Y 47.571,Z 698.605,A -85,B 0,C 180,E1 -30042.814,E2 -30042.814} C_VEL
LIN {X 0,Y 45.678,Z 688.265,A -85,B 0,C 180,E1 -30051.149,E2 -30051.149} C_VEL
LIN {X 0,Y 44.621,Z 674.564,A -85,B 0,C 180,E1 -30060.778,E2 -30060.778} C_VEL
LIN {X 0,Y 44.506,Z 663.914,A -85,B 0,C 180,E1 -30066.802,E2 -30066.802} C_VEL
LIN {X 0,Y 44.729,Z 645.786,A -85,B 0,C 180,E1 -30074.496,E2 -30074.496} C_VEL
LIN {X 0,Y 47.887,Z 587.56,A -85,B 0,C 180,E1 -30095.099,E2 -30095.099} C_VEL
LIN {X 0,Y 46.814,Z 571.364,A -85,B 0,C 180,E1 -30100.167,E2 -30100.167} C_VEL
LIN {X 0,Y 40.1,Z 543.142,A -85,B 0,C 180,E1 -30111.03,E2 -30111.03} C_VEL
LIN {X 0,Y 37.981,Z 535.098,A -85,B 0,C 180,E1 -30115.093,E2 -30115.093} C_VEL
LIN {X 0,Y 36.959,Z 530.996,A -85,B 0,C 180,E1 -30124.667,E2 -30124.667} C_VEL
LIN {X 0,Y 37.112,Z 530.979,A -85,B 0,C 180,E1 -30131.24,E2 -30131.24} C_VEL
LIN {X 0,Y 37.376,Z 530.933,A -85,B 0,C 180,E1 -30141.354,E2 -30141.354} C_VEL
LIN {X 0,Y 36.915,Z 531.011,A -85,B 0,C 180,E1 -30146.217,E2 -30146.217} C_VEL
LIN {X 0,Y 35.062,Z 531.239,A -85,B 0,C 180,E1 -30152.873,E2 -30152.873} C_VEL
LIN {X 0,Y 29.831,Z 531.766,A -85,B 0,C 180,E1 -30173.3,E2 -30173.3} C_VEL
LIN {X 0,Y 29.745,Z 531.769,A -85,B 0,C 180,E1 -30176.021,E2 -30176.021} C_VEL
LIN {X 0,Y 29.838,Z 531.798,A -85,B 0,C 180,E1 -30181.013,E2 -30181.013} C_VEL
LIN {X 0,Y 31.721,Z 538.936,A -85,B 0,C 180,E1 -30191.656,E2 -30191.656} C_VEL
LIN {X 0,Y 35.217,Z 552.016,A -85,B 0,C 180,E1 -30208.01,E2 -30208.01} C_VEL
LIN {X 0,Y 36.355,Z 555.918,A -85,B 0,C 180,E1 -30211.838,E2 -30211.838} C_VEL
LIN {X 0,Y 39.233,Z 588.594,A -85,B 0,C 180,E1 -30223.746,E2 -30223.746} C_VEL
LIN {X 0,Y 42.87,Z 651.416,A -85,B 0,C 180,E1 -30249.139,E2 -30249.139} C_VEL
LIN {X 0,Y 44.62,Z 667.835,A -85,B 0,C 180,E1 -30256,E2 -30256} C_VEL
LIN {X 0,Y 46.451,Z 679.979,A -85,B 0,C 180,E1 -30262.226,E2 -30262.226} C_VEL
LIN {X 0,Y 48.914,Z 690.845,A -85,B 0,C 180,E1 -30269.008,E2 -30269.008} C_VEL
LIN {X 0,Y 51.573,Z 699.117,A -85,B 0,C 180,E1 -30275.151,E2 -30275.151} C_VEL
LIN {X 0,Y 53.941,Z 704.83,A -85,B 0,C 180,E1 -30280.652,E2 -30280.652} C_VEL
LIN {X 0,Y 56.109,Z 708.99,A -85,B 0,C 180,E1 -30285.06,E2 -30285.06} C_VEL
LIN {X 0,Y 56.586,Z 709.804,A -85,B 0,C 180,E1 -30287.051,E2 -30287.051} C_VEL
LIN {X 0,Y 53.306,Z 701.657,A -85,B 0,C 180,E1 -30298.172,E2 -30298.172} C_VEL
LIN {X 0,Y 52.402,Z 692.276,A -85,B 0,C 180,E1 -30309.855,E2 -30309.855} C_VEL
LIN {X 0,Y 53.676,Z 687.179,A -85,B 0,C 180,E1 -30316.748,E2 -30316.748} C_VEL
LIN {X 0,Y 55.841,Z 683.63,A -85,B 0,C 180,E1 -30322.087,E2 -30322.087} C_VEL
LIN {X 0,Y 51.909,Z 687.142,A -85,B 0,C 180,E1 -30327.335,E2 -30327.335} C_VEL
LIN {X 0,Y 48.35,Z 693.013,A -85,B 0,C 180,E1 -30336.05,E2 -30336.05} C_VEL
LIN {X 0,Y 46.943,Z 700.58,A -85,B 0,C 180,E1 -30347.424,E2 -30347.424} C_VEL
LIN {X 0,Y 48.37,Z 708.471,A -85,B 0,C 180,E1 -30359.333,E2 -30359.333} C_VEL
LIN {X 0,Y 52.115,Z 715.911,A -85,B 0,C 180,E1 -30372.4,E2 -30372.4} C_VEL
LIN {X 0,Y 52.486,Z 716.379,A -85,B 0,C 180,E1 -30374.429,E2 -30374.429} C_VEL
LIN {X 0,Y 47.822,Z 708.484,A -85,B 0,C 180,E1 -30383.996,E2 -30383.996} C_VEL
LIN {X 0,Y 44.749,Z 701.113,A -85,B 0,C 180,E1 -30391.89,E2 -30391.89} C_VEL
LIN {X 0,Y 41.92,Z 691.754,A -85,B 0,C 180,E1 -30400.409,E2 -30400.409} C_VEL
LIN {X 0,Y 39.579,Z 678.459,A -85,B 0,C 180,E1 -30411.061,E2 -30411.061} C_VEL
LIN {X 0,Y 38.678,Z 665.598,A -85,B 0,C 180,E1 -30420,E2 -30420} C_VEL
LIN {X 0,Y 38.313,Z 648.59,A -85,B 0,C 180,E1 -30428.903,E2 -30428.903} C_VEL
LIN {X 0,Y 39.985,Z 596.99,A -85,B 0,C 180,E1 -30451.012,E2 -30451.012} C_VEL
LIN {X 0,Y 40.771,Z 587.482,A -85,B 0,C 180,E1 -30454.667,E2 -30454.667} C_VEL
LIN {X 0,Y 39.766,Z 572.375,A -85,B 0,C 180,E1 -30460.223,E2 -30460.223} C_VEL
LIN {X 0,Y 33.12,Z 543.985,A -85,B 0,C 180,E1 -30473.357,E2 -30473.357} C_VEL
LIN {X 0,Y 30.721,Z 534.999,A -85,B 0,C 180,E1 -30479.019,E2 -30479.019} C_VEL
LIN {X 0,Y 29.947,Z 531.757,A -85,B 0,C 180,E1 -30488.576,E2 -30488.576} C_VEL
LIN {X 0,Y 30.141,Z 531.738,A -85,B 0,C 180,E1 -30496.515,E2 -30496.515} C_VEL
LIN {X 0,Y 30.837,Z 531.669,A -85,B 0,C 180,E1 -30509.999,E2 -30509.999} C_VEL
LIN {X 0,Y 30.129,Z 531.739,A -85,B 0,C 180,E1 -30523.488,E2 -30523.488} C_VEL
LIN {X 0,Y 29.745,Z 531.769,A -85,B 0,C 180,E1 -30536.021,E2 -30536.021} C_VEL
LIN {X 0,Y 29.608,Z 532.506,A -85,B 0,C 180,E1 -30540.333,E2 -30540.333} C_VEL
LIN {X 0,Y 29.076,Z 534.917,A -85,B 0,C 180,E1 -30545.193,E2 -30545.193} C_VEL
LIN {X 0,Y 26.408,Z 545.735,A -85,B 0,C 180,E1 -30560.802,E2 -30560.802} C_VEL
LIN {X 0,Y 26.722,Z 547.824,A -85,B 0,C 180,E1 -30564.069,E2 -30564.069} C_VEL
LIN {X 0,Y 29.441,Z 556.137,A -85,B 0,C 180,E1 -30574.86,E2 -30574.86} C_VEL
LIN {X 0,Y 32.808,Z 587.978,A -85,B 0,C 180,E1 -30588.415,E2 -30588.415} C_VEL
LIN {X 0,Y 38.596,Z 650.279,A -85,B 0,C 180,E1 -30616.956,E2 -30616.956} C_VEL
LIN {X 0,Y 40.836,Z 665.397,A -85,B 0,C 180,E1 -30623.453,E2 -30623.453} C_VEL
LIN {X 0,Y 43,Z 677.047,A -85,B 0,C 180,E1 -30629.362,E2 -30629.362} C_VEL
LIN {X 0,Y 46.005,Z 687.784,A -85,B 0,C 180,E1 -30635.941,E2 -30635.941} C_VEL
LIN {X 0,Y 49.004,Z 695.624,A -85,B 0,C 180,E1 -30641.553,E2 -30641.553} C_VEL
LIN {X 0,Y 51.131,Z 700.188,A -85,B 0,C 180,E1 -30645.753,E2 -30645.753} C_VEL
LIN {X 0,Y 51.84,Z 701.544,A -85,B 0,C 180,E1 -30647.325,E2 -30647.325} C_VEL
LIN {X 0,Y 49.147,Z 693.878,A -85,B 0,C 180,E1 -30657.435,E2 -30657.435} C_VEL
LIN {X 0,Y 48.458,Z 687.485,A -85,B 0,C 180,E1 -30665.951,E2 -30665.951} C_VEL
LIN {X 0,Y 49.957,Z 681.13,A -85,B 0,C 180,E1 -30675.269,E2 -30675.269} C_VEL
LIN {X 0,Y 52.279,Z 677.557,A -85,B 0,C 180,E1 -30681.252,E2 -30681.252} C_VEL
LIN {X 0,Y 47.814,Z 681.233,A -85,B 0,C 180,E1 -30687.139,E2 -30687.139} C_VEL
LIN {X 0,Y 43.878,Z 687.295,A -85,B 0,C 180,E1 -30697.03,E2 -30697.03} C_VEL
LIN {X 0,Y 42.379,Z 694.738,A -85,B 0,C 180,E1 -30709.371,E2 -30709.371} C_VEL
LIN {X 0,Y 44.985,Z 705.069,A -85,B 0,C 180,E1 -30726.079,E2 -30726.079} C_VEL
LIN {X 0,Y 46.843,Z 708.587,A -85,B 0,C 180,E1 -30732.461,E2 -30732.461} C_VEL
LIN {X 0,Y 46.2,Z 707.57,A -85,B 0,C 180,E1 -30734.313,E2 -30734.313} C_VEL
LIN {X 0,Y 43.534,Z 702.862,A -85,B 0,C 180,E1 -30739.778,E2 -30739.778} C_VEL
LIN {X 0,Y 40.267,Z 695.647,A -85,B 0,C 180,E1 -30746.946,E2 -30746.946} C_VEL
LIN {X 0,Y 36.802,Z 685.436,A -85,B 0,C 180,E1 -30756.058,E2 -30756.058} C_VEL
LIN {X 0,Y 34.239,Z 672.658,A -85,B 0,C 180,E1 -30766.648,E2 -30766.648} C_VEL
LIN {X 0,Y 32.985,Z 660.367,A -85,B 0,C 180,E1 -30775.417,E2 -30775.417} C_VEL
LIN {X 0,Y 32.21,Z 643.491,A -85,B 0,C 180,E1 -30785.085,E2 -30785.085} C_VEL
LIN {X 0,Y 33.644,Z 587.102,A -85,B 0,C 180,E1 -30814.163,E2 -30814.163} C_VEL
LIN {X 0,Y 32.741,Z 573.411,A -85,B 0,C 180,E1 -30820.229,E2 -30820.229} C_VEL
LIN {X 0,Y 26.323,Z 545.614,A -85,B 0,C 180,E1 -30836.011,E2 -30836.011} C_VEL
LIN {X 0,Y 24.076,Z 537.202,A -85,B 0,C 180,E1 -30842.964,E2 -30842.964} C_VEL
LIN {X 0,Y 23.302,Z 534.834,A -85,B 0,C 180,E1 -30845.546,E2 -30845.546} C_VEL
LIN {X 0,Y 23.02,Z 532.184,A -85,B 0,C 180,E1 -30856.2,E2 -30856.2} C_VEL
LIN {X 0,Y 23.606,Z 532.165,A -85,B 0,C 180,E1 -30869.999,E2 -30869.999} C_VEL
LIN {X 0,Y 22.849,Z 532.188,A -85,B 0,C 180,E1 -30887.913,E2 -30887.913} C_VEL
LIN {X 0,Y 22.69,Z 532.332,A -85,B 0,C 180,E1 -30896.472,E2 -30896.472} C_VEL
LIN {X 0,Y 24.504,Z 539.312,A -85,B 0,C 180,E1 -30910.188,E2 -30910.188} C_VEL
LIN {X 0,Y 26.722,Z 547.824,A -85,B 0,C 180,E1 -30924.069,E2 -30924.069} C_VEL
LIN {X 0,Y 27.319,Z 551.098,A -85,B 0,C 180,E1 -30928.407,E2 -30928.407} C_VEL
LIN {X 0,Y 27.191,Z 556.34,A -85,B 0,C 180,E1 -30934.1,E2 -30934.1} C_VEL
LIN {X 0,Y 26.37,Z 561.732,A -85,B 0,C 180,E1 -30939.275,E2 -30939.275} C_VEL
LIN {X 0,Y 24.98,Z 571.161,A -85,B 0,C 180,E1 -30947.274,E2 -30947.274} C_VEL
LIN {X 0,Y 25.199,Z 577.006,A -85,B 0,C 180,E1 -30950.962,E2 -30950.962} C_VEL
LIN {X 0,Y 26.858,Z 588.395,A -85,B 0,C 180,E1 -30956.25,E2 -30956.25} C_VEL
LIN {X 0,Y 35.141,Z 648.767,A -85,B 0,C 180,E1 -30986.343,E2 -30986.343} C_VEL
LIN {X 0,Y 38.165,Z 663.836,A -85,B 0,C 180,E1 -30992.747,E2 -30992.747} C_VEL
LIN {X 0,Y 41.017,Z 675.551,A -85,B 0,C 180,E1 -30998.481,E2 -30998.481} C_VEL
LIN {X 0,Y 44.937,Z 686.973,A -85,B 0,C 180,E1 -31005.128,E2 -31005.128} C_VEL
LIN {X 0,Y 47.037,Z 691.756,A -85,B 0,C 180,E1 -31008.337,E2 -31008.337} C_VEL
LIN {X 0,Y 45.053,Z 680.77,A -85,B 0,C 180,E1 -31024.003,E2 -31024.003} C_VEL
LIN {X 0,Y 46.668,Z 674.545,A -85,B 0,C 180,E1 -31034.182,E2 -31034.182} C_VEL
LIN {X 0,Y 49.013,Z 671.334,A -85,B 0,C 180,E1 -31040.226,E2 -31040.226} C_VEL
LIN {X 0,Y 44.851,Z 674.251,A -85,B 0,C 180,E1 -31045.507,E2 -31045.507} C_VEL
LIN {X 0,Y 40.464,Z 679.768,A -85,B 0,C 180,E1 -31055.264,E2 -31055.264} C_VEL
LIN {X 0,Y 38.225,Z 687.137,A -85,B 0,C 180,E1 -31068.77,E2 -31068.77} C_VEL
LIN {X 0,Y 40.945,Z 698.983,A -85,B 0,C 180,E1 -31089.251,E2 -31089.251} C_VEL
LIN {X 0,Y 41.129,Z 699.498,A -85,B 0,C 180,E1 -31091.959,E2 -31091.959} C_VEL
LIN {X 0,Y 37.308,Z 692.24,A -85,B 0,C 180,E1 -31098.751,E2 -31098.751} C_VEL
LIN {X 0,Y 33.537,Z 682.92,A -85,B 0,C 180,E1 -31106.627,E2 -31106.627} C_VEL
LIN {X 0,Y 29.952,Z 669.883,A -85,B 0,C 180,E1 -31117.586,E2 -31117.586} C_VEL
LIN {X 0,Y 27.977,Z 657.793,A -85,B 0,C 180,E1 -31126.841,E2 -31126.841} C_VEL
LIN {X 0,Y 26.254,Z 638.237,A -85,B 0,C 180,E1 -31139.52,E2 -31139.52} C_VEL
LIN {X 0,Y 26.6,Z 587.077,A -85,B 0,C 180,E1 -31172.577,E2 -31172.577} C_VEL
LIN {X 0,Y 25.72,Z 574.546,A -85,B 0,C 180,E1 -31179.585,E2 -31179.585} C_VEL
LIN {X 0,Y 19.567,Z 546.92,A -85,B 0,C 180,E1 -31200.618,E2 -31200.618} C_VEL
LIN {X 0,Y 17.798,Z 539.764,A -85,B 0,C 180,E1 -31209.03,E2 -31209.03} C_VEL
LIN {X 0,Y 16.312,Z 534.681,A -85,B 0,C 180,E1 -31217.558,E2 -31217.558} C_VEL
LIN {X 0,Y 16.303,Z 532.63,A -85,B 0,C 180,E1 -31229.998,E2 -31229.998} C_VEL
LIN {X 0,Y 15.908,Z 532.303,A -85,B 0,C 180,E1 -31236.34,E2 -31236.34} C_VEL
LIN {X 0,Y 15.747,Z 532.446,A -85,B 0,C 180,E1 -31247.029,E2 -31247.029} C_VEL
LIN {X 0,Y 17.131,Z 539.129,A -85,B 0,C 180,E1 -31266.502,E2 -31266.502} C_VEL
LIN {X 0,Y 19.348,Z 547.226,A -85,B 0,C 180,E1 -31284.813,E2 -31284.813} C_VEL
LIN {X 0,Y 22.619,Z 556.157,A -85,B 0,C 180,E1 -31299.718,E2 -31299.718} C_VEL
LIN {X 0,Y 23.47,Z 562.804,A -85,B 0,C 180,E1 -31303.417,E2 -31303.417} C_VEL
LIN {X 0,Y 25.199,Z 577.006,A -85,B 0,C 180,E1 -31310.962,E2 -31310.962} C_VEL
LIN {X 0,Y 25.362,Z 582.667,A -85,B 0,C 180,E1 -31314.702,E2 -31314.702} C_VEL
LIN {X 0,Y 24.222,Z 591.652,A -85,B 0,C 180,E1 -31324.166,E2 -31324.166} C_VEL
LIN {X 0,Y 23.651,Z 600.603,A -85,B 0,C 180,E1 -31334.949,E2 -31334.949} C_VEL
LIN {X 0,Y 24.283,Z 606.236,A -85,B 0,C 180,E1 -31339.444,E2 -31339.444} C_VEL
LIN {X 0,Y 33.453,Z 648.966,A -85,B 0,C 180,E1 -31358.107,E2 -31358.107} C_VEL
LIN {X 0,Y 37.004,Z 663.163,A -85,B 0,C 180,E1 -31363.511,E2 -31363.511} C_VEL
LIN {X 0,Y 40.6,Z 675.258,A -85,B 0,C 180,E1 -31368.801,E2 -31368.801} C_VEL
LIN {X 0,Y 42.353,Z 679.838,A -85,B 0,C 180,E1 -31371.152,E2 -31371.152} C_VEL
LIN {X 0,Y 42.239,Z 678.569,A -85,B 0,C 180,E1 -31374.378,E2 -31374.378} C_VEL
LIN {X 0,Y 42.457,Z 671.065,A -85,B 0,C 180,E1 -31386.963,E2 -31386.963} C_VEL
LIN {X 0,Y 44.941,Z 666.016,A -85,B 0,C 180,E1 -31396.637,E2 -31396.637} C_VEL
LIN {X 0,Y 45.936,Z 664.983,A -85,B 0,C 180,E1 -31399.327,E2 -31399.327} C_VEL
LIN {X 0,Y 42.434,Z 667.139,A -85,B 0,C 180,E1 -31403.578,E2 -31403.578} C_VEL
LIN {X 0,Y 37.839,Z 671.729,A -85,B 0,C 180,E1 -31412.37,E2 -31412.37} C_VEL
LIN {X 0,Y 34.807,Z 677.693,A -85,B 0,C 180,E1 -31424.62,E2 -31424.62} C_VEL
LIN {X 0,Y 35.026,Z 687.052,A -85,B 0,C 180,E1 -31443.491,E2 -31443.491} C_VEL
LIN {X 0,Y 35.941,Z 689.757,A -85,B 0,C 180,E1 -31448.54,E2 -31448.54} C_VEL
LIN {X 0,Y 31.37,Z 680.304,A -85,B 0,C 180,E1 -31455.564,E2 -31455.564} C_VEL
LIN {X 0,Y 26.736,Z 666.731,A -85,B 0,C 180,E1 -31466.04,E2 -31466.04} C_VEL
LIN {X 0,Y 24.357,Z 656.393,A -85,B 0,C 180,E1 -31473.779,E2 -31473.779} C_VEL
LIN {X 0,Y 21.301,Z 637.058,A -85,B 0,C 180,E1 -31487.485,E2 -31487.485} C_VEL
LIN {X 0,Y 19.534,Z 586.46,A -85,B 0,C 180,E1 -31530.277,E2 -31530.277} C_VEL
LIN {X 0,Y 18.599,Z 575.24,A -85,B 0,C 180,E1 -31538.795,E2 -31538.795} C_VEL
LIN {X 0,Y 13.175,Z 549.385,A -85,B 0,C 180,E1 -31567.454,E2 -31567.454} C_VEL
LIN {X 0,Y 11.898,Z 542.433,A -85,B 0,C 180,E1 -31580.435,E2 -31580.435} C_VEL
LIN {X 0,Y 10.806,Z 537.366,A -85,B 0,C 180,E1 -31595.131,E2 -31595.131} C_VEL
LIN {X 0,Y 9.415,Z 537.206,A -85,B 0,C 180,E1 -31609.181,E2 -31609.181} C_VEL
LIN {X 0,Y 10.586,Z 542.142,A -85,B 0,C 180,E1 -31631.593,E2 -31631.593} C_VEL
LIN {X 0,Y 14.677,Z 552.864,A -85,B 0,C 180,E1 -31663.271,E2 -31663.271} C_VEL
LIN {X 0,Y 16.108,Z 555.786,A -85,B 0,C 180,E1 -31669.011,E2 -31669.011} C_VEL
LIN {X 0,Y 16.946,Z 560.09,A -85,B 0,C 180,E1 -31671.747,E2 -31671.747} C_VEL
LIN {X 0,Y 21.595,Z 587.625,A -85,B 0,C 180,E1 -31687.476,E2 -31687.476} C_VEL
LIN {X 0,Y 24.283,Z 606.236,A -85,B 0,C 180,E1 -31699.444,E2 -31699.444} C_VEL
LIN {X 0,Y 25.072,Z 611.789,A -85,B 0,C 180,E1 -31703.644,E2 -31703.644} C_VEL
LIN {X 0,Y 27.841,Z 629.239,A -85,B 0,C 180,E1 -31723.335,E2 -31723.335} C_VEL
LIN {X 0,Y 29.301,Z 634.744,A -85,B 0,C 180,E1 -31726.686,E2 -31726.686} C_VEL
LIN {X 0,Y 35.422,Z 656.407,A -85,B 0,C 180,E1 -31732.527,E2 -31732.527} C_VEL
LIN {X 0,Y 39.045,Z 667.849,A -85,B 0,C 180,E1 -31736.36,E2 -31736.36} C_VEL
LIN {X 0,Y 39.28,Z 667.824,A -85,B 0,C 180,E1 -31737.879,E2 -31737.879} C_VEL
LIN {X 0,Y 40.885,Z 661.306,A -85,B 0,C 180,E1 -31751.173,E2 -31751.173} C_VEL
LIN {X 0,Y 43.241,Z 658.477,A -85,B 0,C 180,E1 -31758.368,E2 -31758.368} C_VEL
LIN {X 0,Y 39.8,Z 660.331,A -85,B 0,C 180,E1 -31762.39,E2 -31762.39} C_VEL
LIN {X 0,Y 34.402,Z 665.206,A -85,B 0,C 180,E1 -31772.607,E2 -31772.607} C_VEL
LIN {X 0,Y 31.007,Z 672.136,A -85,B 0,C 180,E1 -31788.81,E2 -31788.81} C_VEL
LIN {X 0,Y 30.882,Z 677.349,A -85,B 0,C 180,E1 -31800.801,E2 -31800.801} C_VEL
LIN {X 0,Y 29.825,Z 675.841,A -85,B 0,C 180,E1 -31804.437,E2 -31804.437} C_VEL
LIN {X 0,Y 24.866,Z 663.453,A -85,B 0,C 180,E1 -31812.103,E2 -31812.103} C_VEL
LIN {X 0,Y 21.715,Z 652.431,A -85,B 0,C 180,E1 -31818.897,E2 -31818.897} C_VEL
LIN {X 0,Y 15.936,Z 625.897,A -85,B 0,C 180,E1 -31837.3,E2 -31837.3} C_VEL
LIN {X 0,Y 12.67,Z 586.565,A -85,B 0,C 180,E1 -31883.895,E2 -31883.895} C_VEL
LIN {X 0,Y 11.622,Z 576.332,A -85,B 0,C 180,E1 -31895.649,E2 -31895.649} C_VEL
LIN {X 0,Y 7.173,Z 549.877,A -85,B 0,C 180,E1 -31951.418,E2 -31951.418} C_VEL
LIN {X 0,Y 7.17,Z 546.964,A -85,B 0,C 180,E1 -31961.445,E2 -31961.445} C_VEL
LIN {X 0,Y 6.33,Z 547.644,A -85,B 0,C 180,E1 -31972.838,E2 -31972.838} C_VEL
LIN {X 0,Y 5.814,Z 550.118,A -85,B 0,C 180,E1 -32017.207,E2 -32017.207} C_VEL
LIN {X 0,Y 7.041,Z 550.549,A -85,B 0,C 180,E1 -32036.461,E2 -32036.461} C_VEL
LIN {X 0,Y 7.424,Z 550.664,A -85,B 0,C 180,E1 -32039.242,E2 -32039.242} C_VEL
LIN {X 0,Y 10.832,Z 556.173,A -85,B 0,C 180,E1 -32049.81,E2 -32049.81} C_VEL
LIN {X 0,Y 12.041,Z 561.188,A -85,B 0,C 180,E1 -32052.395,E2 -32052.395} C_VEL
LIN {X 0,Y 17.765,Z 586.677,A -85,B 0,C 180,E1 -32064.857,E2 -32064.857} C_VEL
LIN {X 0,Y 29.301,Z 634.744,A -85,B 0,C 180,E1 -32086.686,E2 -32086.686} C_VEL
LIN {X 0,Y 30.318,Z 638.369,A -85,B 0,C 180,E1 -32089.209,E2 -32089.209} C_VEL
LIN {X 0,Y 34.649,Z 649.132,A -85,B 0,C 180,E1 -32101.381,E2 -32101.381} C_VEL
LIN {X 0,Y 36.001,Z 652.754,A -85,B 0,C 180,E1 -32102.953,E2 -32102.953} C_VEL
LIN {X 0,Y 37.384,Z 656.864,A -85,B 0,C 180,E1 -32103.87,E2 -32103.87} C_VEL
LIN {X 0,Y 39.449,Z 652.927,A -85,B 0,C 180,E1 -32114.033,E2 -32114.033} C_VEL
LIN {X 0,Y 40.703,Z 651.896,A -85,B 0,C 180,E1 -32117.522,E2 -32117.522} C_VEL
LIN {X 0,Y 35.989,Z 654.373,A -85,B 0,C 180,E1 -32123.318,E2 -32123.318} C_VEL
LIN {X 0,Y 30.1,Z 660.034,A -85,B 0,C 180,E1 -32136.736,E2 -32136.736} C_VEL
LIN {X 0,Y 28.021,Z 664.337,A -85,B 0,C 180,E1 -32148.276,E2 -32148.276} C_VEL
LIN {X 0,Y 27.077,Z 665.556,A -85,B 0,C 180,E1 -32155.051,E2 -32155.051} C_VEL
LIN {X 0,Y 22.708,Z 653.875,A -85,B 0,C 180,E1 -32159.488,E2 -32159.488} C_VEL
LIN {X 0,Y 16.996,Z 634.9,A -85,B 0,C 180,E1 -32166.366,E2 -32166.366} C_VEL
LIN {X 0,Y 6.326,Z 586.348,A -85,B 0,C 180,E1 -32223.221,E2 -32223.221} C_VEL
LIN {X 0,Y 4.714,Z 577.122,A -85,B 0,C 180,E1 -32242.507,E2 -32242.507} C_VEL
LIN {X 0,Y 3.572,Z 557.182,A -85,B 0,C 180,E1 -32361.041,E2 -32361.041} C_VEL
LIN {X 0,Y 3.874,Z 557.03,A -85,B 0,C 180,E1 -32375.517,E2 -32375.517} C_VEL
LIN {X 0,Y 4.584,Z 560.021,A -85,B 0,C 180,E1 -32406.166,E2 -32406.166} C_VEL
LIN {X 0,Y 8.022,Z 569.164,A -85,B 0,C 180,E1 -32441.454,E2 -32441.454} C_VEL
LIN {X 0,Y 11.018,Z 573.015,A -85,B 0,C 180,E1 -32447.649,E2 -32447.649} C_VEL
LIN {X 0,Y 13.19,Z 574.153,A -85,B 0,C 180,E1 -32448.529,E2 -32448.529} C_VEL
LIN {X 0,Y 16.659,Z 586.957,A -85,B 0,C 180,E1 -32448.718,E2 -32448.718} C_VEL
LIN {X 0,Y 32.792,Z 642.497,A -85,B 0,C 180,E1 -32461.469,E2 -32461.469} C_VEL
LIN {X 0,Y 36.001,Z 652.754,A -85,B 0,C 180,E1 -32462.953,E2 -32462.953} C_VEL
LIN {X 0,Y 35.965,Z 653.896,A -85,B 0,C 180,E1 -32464.099,E2 -32464.099} C_VEL
LIN {X 0,Y 34.963,Z 654.761,A -85,B 0,C 180,E1 -32467.673,E2 -32467.673} C_VEL
LIN {X 0,Y 33.091,Z 654.546,A -85,B 0,C 180,E1 -32473.582,E2 -32473.582} C_VEL
LIN {X 0,Y 29.122,Z 652.593,A -85,B 0,C 180,E1 -32488.507,E2 -32488.507} C_VEL
LIN {X 0,Y 27.851,Z 652.738,A -85,B 0,C 180,E1 -32494.63,E2 -32494.63} C_VEL
LIN {X 0,Y 26.941,Z 653.623,A -85,B 0,C 180,E1 -32498.972,E2 -32498.972} C_VEL
LIN {X 0,Y 26.412,Z 654.474,A -85,B 0,C 180,E1 -32501.531,E2 -32501.531} C_VEL
LIN {X 0,Y 25.779,Z 654.397,A -85,B 0,C 180,E1 -32503.641,E2 -32503.641} C_VEL
LIN {X 0,Y 19.328,Z 634.727,A -85,B 0,C 180,E1 -32505.016,E2 -32505.016} C_VEL
LIN {X 0,Y 4.489,Z 585.781,A -85,B 0,C 180,E1 -32502.703,E2 -32502.703} C_VEL
LIN {X 0,Y 3.246,Z 577.871,A -85,B 0,C 180,E1 -32477.549,E2 -32477.549} C_VEL
LIN {X 0,Y 3.444,Z 575.845,A -85,B 0,C 180,E1 -32465.798,E2 -32465.798} C_VEL
LIN {X 0,Y 4.511,Z 576.09,A -85,B 0,C 180,E1 -32461.602,E2 -32461.602} C_VEL
LIN {X 0,Y 7.768,Z 579.296,A -85,B 0,C 180,E1 -32460.888,E2 -32460.888} C_VEL
LIN {X 0,Y 17.914,Z 603.252,A -85,B 0,C 180,E1 -32472.995,E2 -32472.995} C_VEL
LIN {X 0,Y 23.732,Z 614.525,A -85,B 0,C 180,E1 -32473.782,E2 -32473.782} C_VEL
LIN {X 0,Y 26.495,Z 618.55,A -85,B 0,C 180,E1 -32473.378,E2 -32473.378} C_VEL
LIN {X 0,Y 27.872,Z 619.398,A -85,B 0,C 180,E1 -32472.515,E2 -32472.515} C_VEL
LIN {X 0,Y 28.353,Z 619.403,A -85,B 0,C 180,E1 -32472.063,E2 -32472.063} C_VEL
LIN {X 0,Y 36.808,Z 646.217,A -85,B 0,C 180,E1 -32472.689,E2 -32472.689} C_VEL
LIN {X 0,Y 38.069,Z 645.313,A -85,B 0,C 180,E1 -32476.788,E2 -32476.788} C_VEL
LIN {X 0,Y 32.809,Z 648.006,A -85,B 0,C 180,E1 -32483.678,E2 -32483.678} C_VEL
LIN {X 0,Y 26.941,Z 653.623,A -85,B 0,C 180,E1 -32498.972,E2 -32498.972} C_VEL
LIN {X 0,Y 26.531,Z 652.705,A -85,B 0,C 180,E1 -32499.286,E2 -32499.286} C_VEL
LIN {X 0,Y 26.526,Z 649.643,A -85,B 0,C 180,E1 -32496.35,E2 -32496.35} C_VEL
LIN {X 0,Y 28.379,Z 640.041,A -85,B 0,C 180,E1 -32484.962,E2 -32484.962} C_VEL
LIN {X 0,Y 28.417,Z 636.54,A -85,B 0,C 180,E1 -32482.57,E2 -32482.57} C_VEL
LIN {X 0,Y 27.684,Z 633.94,A -85,B 0,C 180,E1 -32481.903,E2 -32481.903} C_VEL
LIN {X 0,Y 23.748,Z 624.289,A -85,B 0,C 180,E1 -32481.016,E2 -32481.016} C_VEL
LIN {X 0,Y 20.847,Z 620.83,A -85,B 0,C 180,E1 -32483.73,E2 -32483.73} C_VEL
LIN {X 0,Y 18.554,Z 617.067,A -85,B 0,C 180,E1 -32485.491,E2 -32485.491} C_VEL
LIN {X 0,Y 26.721,Z 643.954,A -85,B 0,C 180,E1 -32490.941,E2 -32490.941} C_VEL
LIN {X 0,Y 30.504,Z 641.109,A -85,B 0,C 180,E1 -32482.598,E2 -32482.598} C_VEL
LIN {X 0,Y 27.684,Z 633.94,A -85,B 0,C 180,E1 -32481.903,E2 -32481.903} C_VEL
LIN {X 0,Y 27.684,Z 633.94,A -85,B 0,C 180,E1 -32481.903,E2 -32481.903}

QRS_NEXT_CUT()

QRS_NEXT()
QRS_HOME()

END
